C01778=1030.440,193.535,-110.316,169.514,44.801,158.470
C01779=1030.433,193.286,-110.292,169.510,44.803,158.470
C01780=1030.427,193.037,-110.268,169.506,44.804,158.470
C01781=1030.422,192.789,-110.244,169.503,44.807,158.470
C01782=1030.415,192.540,-110.220,169.500,44.809,158.470
C01783=1030.410,192.291,-110.196,169.497,44.811,158.470
C01784=1030.403,192.042,-110.171,169.493,44.812,158.470
C01785=1030.398,191.794,-110.147,169.489,44.814,158.471
C01786=1030.391,191.545,-110.123,169.486,44.817,158.471
C01787=1030.386,191.296,-110.099,169.483,44.818,158.471
C01788=1030.380,191.048,-110.075,169.479,44.820,158.471
C01789=1030.374,190.799,-110.051,169.476,44.822,158.471
C01790=1030.368,190.550,-110.027,169.472,44.824,158.471
C01791=1030.361,190.301,-110.003,169.469,44.826,158.471
C01792=1030.356,190.053,-109.979,169.466,44.828,158.471
C01793=1030.349,189.804,-109.955,169.462,44.830,158.471
C01794=1030.344,189.555,-109.930,169.459,44.831,158.471
C01795=1030.338,189.306,-109.907,169.455,44.834,158.471
C01796=1030.332,189.057,-109.883,169.451,44.836,158.471
C01797=1030.325,188.774,-109.856,169.448,44.838,158.471
C01798=1030.319,188.491,-109.828,169.444,44.840,158.471
C01799=1030.312,188.207,-109.801,169.441,44.842,158.471
C01800=1030.305,187.923,-109.774,169.436,44.845,158.471
C01801=1030.299,187.675,-109.750,169.433,44.847,158.472
C01802=1030.293,187.426,-109.725,169.430,44.848,158.472
C01803=1030.288,187.177,-109.702,169.426,44.850,158.472
C01804=1030.282,186.929,-109.679,169.423,44.852,158.472
C01805=1030.276,186.679,-109.654,169.420,44.854,158.472
C01806=1030.270,186.431,-109.631,169.416,44.856,158.472
C01807=1030.264,186.182,-109.606,169.413,44.858,158.472
C01808=1030.258,185.933,-109.583,169.409,44.860,158.472
C01809=1030.252,185.685,-109.559,169.407,44.862,158.472
C01810=1030.247,185.436,-109.535,169.403,44.864,158.472
C01811=1030.240,185.186,-109.512,169.399,44.866,158.472
C01812=1030.235,184.938,-109.487,169.396,44.868,158.472
C01813=1030.229,184.689,-109.464,169.393,44.870,158.472
C01814=1030.223,184.440,-109.439,169.390,44.872,158.472
C01815=1030.217,184.191,-109.416,169.386,44.874,158.472
C01816=1030.211,183.943,-109.393,169.383,44.875,158.473
C01817=1030.206,183.694,-109.369,169.380,44.878,158.473
C01818=1030.200,183.445,-109.345,169.376,44.880,158.473
C01819=1030.194,183.196,-109.321,169.373,44.881,158.473
C01820=1030.189,182.947,-109.298,169.370,44.883,158.473
C01821=1030.183,182.699,-109.274,169.366,44.885,158.473
C01822=1030.176,182.449,-109.251,169.363,44.888,158.473
C01823=1030.170,182.201,-109.227,169.360,44.890,158.473
C01824=1030.164,181.953,-109.205,169.357,44.892,158.473
C01825=1030.158,181.703,-109.182,169.353,44.895,158.473
C01826=1030.152,181.455,-109.158,169.350,44.897,158.474
C01827=1030.146,181.206,-109.135,169.347,44.899,158.474
C01828=1030.139,180.956,-109.112,169.344,44.901,158.474
C01829=1030.133,180.708,-109.088,169.340,44.903,158.474
C01830=1030.127,180.459,-109.066,169.336,44.905,158.474
C01831=1030.121,180.210,-109.042,169.333,44.907,158.474
C01832=1030.115,179.962,-109.019,169.330,44.909,158.474
C01833=1030.109,179.713,-108.996,169.327,44.912,158.474
C01834=1030.103,179.464,-108.973,169.323,44.914,158.475
C01835=1030.096,179.215,-108.949,169.320,44.916,158.475
C01836=1030.090,178.966,-108.926,169.317,44.918,158.475
C01837=1030.084,178.717,-108.903,169.314,44.921,158.475
C01838=1030.079,178.468,-108.880,169.310,44.923,158.475
C01839=1030.072,178.219,-108.856,169.308,44.925,158.475
C01840=1030.065,177.971,-108.834,169.304,44.927,158.475
C01841=1030.060,177.722,-108.811,169.301,44.930,158.475
C01842=1030.054,177.473,-108.788,169.297,44.932,158.476
C01843=1030.048,177.223,-108.765,169.295,44.934,158.476
C01844=1030.042,176.975,-108.741,169.291,44.936,158.476
C01845=1030.035,176.727,-108.719,169.288,44.938,158.476
C01846=1030.029,176.478,-108.696,169.285,44.940,158.476
C01847=1030.024,176.229,-108.673,169.281,44.942,158.476
C01848=1030.017,175.979,-108.650,169.278,44.945,158.476
C01849=1030.012,175.730,-108.627,169.276,44.947,158.476
C01850=1030.005,175.482,-108.604,169.272,44.949,158.477
C01851=1029.999,175.233,-108.581,169.268,44.951,158.477
C01852=1029.993,174.984,-108.558,169.265,44.954,158.477
C01853=1029.988,174.736,-108.535,169.262,44.956,158.477
C01854=1029.981,174.486,-108.512,169.259,44.958,158.477
C01855=1029.975,174.237,-108.489,169.255,44.961,158.477
C01856=1029.969,173.989,-108.466,169.253,44.963,158.477
C01857=1029.963,173.740,-108.443,169.249,44.965,158.477
C01858=1029.958,173.491,-108.420,169.247,44.967,158.478
C01859=1029.951,173.242,-108.398,169.243,44.969,158.478
C01860=1029.945,172.993,-108.375,169.240,44.971,158.478
C01861=1029.938,172.709,-108.349,169.236,44.974,158.478
C01862=1029.931,172.426,-108.322,169.233,44.976,158.478
C01863=1029.926,172.142,-108.296,169.229,44.979,158.478
C01864=1029.918,171.858,-108.270,169.226,44.981,158.478
C01865=1029.912,171.609,-108.248,169.222,44.983,158.478
C01866=1029.906,171.360,-108.225,169.219,44.986,158.479
C01867=1029.900,171.111,-108.202,169.216,44.988,158.479
C01868=1029.895,170.862,-108.179,169.213,44.990,158.479
C01869=1029.888,170.614,-108.156,169.210,44.992,158.479
C01870=1029.882,170.365,-108.133,169.207,44.994,158.479
C01871=1029.877,170.116,-108.110,169.203,44.996,158.479
C01872=1029.870,169.866,-108.087,169.201,44.999,158.480
C01873=1029.864,169.618,-108.065,169.197,45.001,158.480
C01874=1029.859,169.368,-108.043,169.195,45.003,158.480
C01875=1029.853,169.119,-108.020,169.191,45.005,158.480
C01876=1029.847,168.871,-107.997,169.188,45.008,158.480
C01877=1029.841,168.622,-107.974,169.185,45.010,158.480
C01878=1029.835,168.373,-107.951,169.182,45.012,158.480
C01879=1029.829,168.124,-107.928,169.179,45.014,158.480
C01880=1029.823,167.875,-107.906,169.176,45.017,158.480
C01881=1029.818,167.626,-107.883,169.173,45.019,158.481
C01882=1029.812,167.377,-107.861,169.170,45.021,158.481
C01883=1029.806,167.128,-107.838,169.166,45.023,158.481
C01884=1029.801,166.880,-107.815,169.164,45.025,158.481
C01885=1029.794,166.632,-107.793,169.160,45.028,158.481
C01886=1029.788,166.383,-107.770,169.158,45.030,158.481
C01887=1029.783,166.134,-107.747,169.154,45.032,158.481
C01888=1029.777,165.884,-107.725,169.152,45.034,158.482
C01889=1029.771,165.636,-107.703,169.148,45.037,158.482
C01890=1029.765,165.387,-107.680,169.146,45.039,158.482
C01891=1029.759,165.138,-107.657,169.142,45.041,158.482
C01892=1029.754,164.888,-107.634,169.140,45.043,158.482
C01893=1029.747,164.640,-107.612,169.136,45.045,158.482
C01894=1029.742,164.391,-107.589,169.133,45.047,158.482
C01895=1029.736,164.142,-107.566,169.130,45.050,158.483
C01896=1029.731,163.892,-107.544,169.128,45.052,158.483
C01897=1029.725,163.645,-107.522,169.124,45.054,158.483
C01898=1029.719,163.396,-107.499,169.121,45.056,158.483
C01899=1029.714,163.146,-107.477,169.118,45.058,158.483
C01900=1029.707,162.898,-107.454,169.116,45.061,158.483
C01901=1029.701,162.649,-107.432,169.112,45.063,158.483
C01902=1029.696,162.399,-107.409,169.110,45.065,158.484
C01903=1029.690,162.150,-107.386,169.106,45.067,158.484
C01904=1029.684,161.902,-107.364,169.103,45.069,158.484
C01905=1029.679,161.653,-107.342,169.100,45.071,158.484
C01906=1029.673,161.404,-107.319,169.098,45.074,158.484
C01907=1029.667,161.155,-107.296,169.094,45.076,158.484
C01908=1029.661,160.906,-107.275,169.092,45.078,158.484
C01909=1029.656,160.657,-107.252,169.088,45.080,158.484
C01910=1029.650,160.407,-107.229,169.085,45.082,158.485
C01911=1029.644,160.160,-107.207,169.082,45.085,158.485
C01912=1029.639,159.911,-107.185,169.080,45.087,158.485
C01913=1029.633,159.661,-107.162,169.076,45.089,158.485
C01914=1029.627,159.413,-107.140,169.073,45.091,158.485
C01915=1029.621,159.163,-107.118,169.070,45.094,158.485
C01916=1029.615,158.914,-107.096,169.068,45.096,158.486
C01917=1029.609,158.666,-107.074,169.064,45.099,158.486
C01918=1029.603,158.417,-107.052,169.062,45.101,158.486
C01919=1029.597,158.168,-107.029,169.058,45.103,158.486
C01920=1029.591,157.919,-107.008,169.056,45.106,158.486
C01921=1029.585,157.669,-106.986,169.052,45.108,158.486
C01922=1029.579,157.420,-106.963,169.050,45.110,158.487
C01923=1029.573,157.171,-106.942,169.046,45.113,158.487
C01924=1029.568,156.923,-106.920,169.044,45.115,158.487
C01925=1029.558,156.533,-106.886,169.039,45.118,158.487
C01926=1029.548,156.143,-106.851,169.035,45.122,158.487
C01927=1029.539,155.754,-106.817,169.030,45.126,158.488
C01928=1029.530,155.363,-106.782,169.026,45.130,158.488
C01929=1029.525,155.115,-106.761,169.022,45.132,158.488
C01930=1029.518,154.866,-106.739,169.020,45.134,158.488
C01931=1029.513,154.617,-106.716,169.016,45.137,158.489
C01932=1029.506,154.368,-106.695,169.014,45.139,158.489
C01933=1029.500,154.118,-106.673,169.010,45.142,158.489
C01934=1029.495,153.870,-106.652,169.008,45.144,158.489
C01935=1029.489,153.620,-106.629,169.004,45.147,158.489
C01936=1029.483,153.372,-106.607,169.002,45.149,158.489
C01937=1029.477,153.123,-106.585,168.999,45.151,158.490
C01938=1029.471,152.874,-106.564,168.996,45.153,158.490
C01939=1029.465,152.625,-106.543,168.994,45.155,158.490
C01940=1029.459,152.376,-106.521,168.990,45.158,158.490
C01941=1029.450,151.983,-106.487,168.986,45.162,158.490
C01942=1029.440,151.591,-106.452,168.981,45.166,158.491
C01943=1029.431,151.198,-106.419,168.977,45.170,158.491
C01944=1029.422,150.805,-106.384,168.972,45.174,158.491
C01945=1029.416,150.556,-106.362,168.969,45.176,158.491
C01946=1029.410,150.308,-106.340,168.966,45.178,158.492
C01947=1029.404,150.059,-106.319,168.964,45.180,158.492
C01948=1029.398,149.810,-106.297,168.960,45.183,158.492
C01949=1029.392,149.561,-106.276,168.958,45.185,158.492
C01950=1029.386,149.312,-106.254,168.955,45.188,158.492
C01951=1029.380,149.063,-106.232,168.952,45.190,158.493
C01952=1029.374,148.814,-106.211,168.950,45.193,158.493
C01953=1029.368,148.565,-106.190,168.946,45.195,158.493
C01954=1029.362,148.316,-106.168,168.944,45.198,158.493
C01955=1029.356,148.068,-106.147,168.940,45.200,158.493
C01956=1029.351,147.818,-106.124,168.938,45.202,158.494
C01957=1029.345,147.569,-106.103,168.935,45.204,158.494
C01958=1029.339,147.320,-106.082,168.932,45.207,158.494
C01959=1029.333,147.071,-106.061,168.929,45.209,158.494
C01960=1029.327,146.821,-106.039,168.926,45.212,158.494
C01961=1029.321,146.573,-106.018,168.924,45.214,158.494
C01962=1029.315,146.324,-105.996,168.920,45.217,158.495
C01963=1029.308,146.075,-105.975,168.918,45.219,158.495
C01964=1029.303,145.826,-105.954,168.916,45.222,158.495
C01965=1029.297,145.577,-105.932,168.912,45.224,158.495
C01966=1029.291,145.328,-105.911,168.910,45.226,158.495
C01967=1029.285,145.079,-105.890,168.906,45.229,158.496
C01968=1029.279,144.829,-105.868,168.904,45.231,158.496
C01969=1029.273,144.580,-105.847,168.901,45.234,158.496
C01970=1029.267,144.332,-105.826,168.898,45.237,158.496
C01971=1029.260,144.083,-105.804,168.896,45.239,158.496
C01972=1029.255,143.834,-105.784,168.892,45.242,158.497
C01973=1029.249,143.585,-105.762,168.890,45.244,158.497
C01974=1029.243,143.335,-105.741,168.887,45.247,158.497
C01975=1029.237,143.087,-105.719,168.884,45.249,158.497
C01976=1029.231,142.837,-105.699,168.881,45.251,158.497
C01977=1029.225,142.589,-105.678,168.878,45.254,158.498
C01978=1029.219,142.340,-105.656,168.876,45.256,158.498
C01979=1029.213,142.090,-105.634,168.873,45.259,158.498
C01980=1029.208,141.841,-105.614,168.870,45.262,158.498
C01981=1029.201,141.592,-105.592,168.867,45.264,158.498
C01982=1029.195,141.344,-105.572,168.864,45.266,158.499
C01983=1029.189,141.094,-105.551,168.862,45.268,158.499
C01984=1029.184,140.846,-105.529,168.859,45.271,158.499
C01985=1029.176,140.561,-105.505,168.855,45.274,158.499
C01986=1029.170,140.276,-105.480,168.853,45.277,158.500
C01987=1029.163,139.991,-105.457,168.850,45.280,158.500
C01988=1029.157,139.707,-105.433,168.846,45.283,158.500
C01989=1029.151,139.458,-105.411,168.844,45.285,158.500
C01990=1029.145,139.209,-105.391,168.841,45.287,158.500
C01991=1029.139,138.959,-105.369,168.838,45.289,158.501
C01992=1029.133,138.711,-105.349,168.835,45.292,158.501
C01993=1029.127,138.461,-105.327,168.832,45.295,158.501
C01994=1029.121,138.213,-105.306,168.830,45.297,158.501
C01995=1029.115,137.963,-105.286,168.827,45.300,158.501
C01996=1029.109,137.715,-105.264,168.824,45.302,158.502
C01997=1029.103,137.465,-105.244,168.822,45.304,158.502
C01998=1029.097,137.217,-105.223,168.818,45.307,158.502
C01999=1029.091,136.967,-105.202,168.816,45.310,158.502
C02000=1029.086,136.719,-105.181,168.813,45.312,158.502
C02001=1029.079,136.469,-105.160,168.810,45.315,158.503
C02002=1029.074,136.221,-105.139,168.808,45.318,158.503
C02003=1029.067,135.971,-105.119,168.805,45.320,158.503
C02004=1029.061,135.722,-105.097,168.802,45.322,158.503
C02005=1029.056,135.473,-105.077,168.800,45.325,158.504
C02006=1029.050,135.224,-105.057,168.797,45.328,158.504
C02007=1029.043,134.975,-105.035,168.794,45.330,158.504
C02008=1029.037,134.726,-105.015,168.791,45.333,158.504
C02009=1029.031,134.477,-104.993,168.789,45.335,158.504
C02010=1029.026,134.228,-104.973,168.786,45.337,158.505
C02011=1029.019,133.978,-104.952,168.783,45.340,158.505
C02012=1029.014,133.729,-104.931,168.780,45.343,158.505
C02013=1029.007,133.480,-104.911,168.778,45.345,158.505
C02014=1029.002,133.231,-104.890,168.775,45.348,158.505
C02015=1028.996,132.983,-104.870,168.772,45.351,158.506
C02016=1028.990,132.733,-104.849,168.770,45.353,158.506
C02017=1028.983,132.485,-104.828,168.766,45.355,158.506
C02018=1028.978,132.235,-104.807,168.764,45.358,158.506
C02019=1028.972,131.986,-104.787,168.762,45.360,158.506
C02020=1028.965,131.737,-104.766,168.758,45.363,158.507
C02021=1028.960,131.488,-104.745,168.756,45.366,158.507
C02022=1028.954,131.239,-104.725,168.754,45.368,158.507
C02023=1028.948,130.990,-104.703,168.750,45.370,158.507
C02024=1028.942,130.741,-104.683,168.748,45.373,158.508
C02025=1028.936,130.491,-104.663,168.745,45.375,158.508
C02026=1028.930,130.242,-104.643,168.742,45.378,158.508
C02027=1028.924,129.993,-104.623,168.740,45.381,158.508
C02028=1028.918,129.744,-104.601,168.738,45.383,158.509
C02029=1028.912,129.495,-104.581,168.734,45.386,158.509
C02030=1028.905,129.246,-104.561,168.732,45.389,158.509
C02031=1028.899,128.997,-104.541,168.729,45.392,158.509
C02032=1028.894,128.747,-104.520,168.726,45.394,158.509
C02033=1028.888,128.498,-104.500,168.724,45.396,158.510
C02034=1028.882,128.250,-104.480,168.721,45.399,158.510
C02035=1028.875,128.000,-104.460,168.718,45.402,158.510
C02036=1028.869,127.752,-104.438,168.716,45.405,158.510
C02037=1028.863,127.503,-104.418,168.713,45.408,158.511
C02038=1028.857,127.253,-104.398,168.710,45.410,158.511
C02039=1028.851,127.004,-104.378,168.708,45.412,158.511
C02040=1028.844,126.755,-104.358,168.705,45.415,158.511
C02041=1028.839,126.506,-104.337,168.702,45.418,158.512
C02042=1028.833,126.257,-104.317,168.700,45.420,158.512
C02043=1028.826,126.007,-104.297,168.696,45.423,158.512
C02044=1028.820,125.759,-104.277,168.694,45.425,158.512
C02045=1028.815,125.510,-104.256,168.691,45.428,158.512
C02046=1028.809,125.260,-104.236,168.689,45.431,158.513
C02047=1028.803,125.011,-104.216,168.686,45.434,158.513
C02048=1028.797,124.762,-104.196,168.684,45.436,158.513
C02049=1028.790,124.477,-104.172,168.681,45.439,158.514
C02050=1028.782,124.193,-104.150,168.677,45.442,158.514
C02051=1028.776,123.908,-104.127,168.674,45.445,158.514
C02052=1028.769,123.624,-104.104,168.671,45.448,158.514
C02053=1028.763,123.374,-104.083,168.669,45.451,158.515
C02054=1028.757,123.125,-104.063,168.666,45.453,158.515
C02055=1028.751,122.876,-104.043,168.663,45.456,158.515
C02056=1028.744,122.627,-104.023,168.661,45.459,158.515
C02057=1028.738,122.378,-104.003,168.658,45.461,158.515
C02058=1028.733,122.129,-103.982,168.655,45.464,158.516
C02059=1028.727,121.880,-103.962,168.653,45.466,158.516
C02060=1028.721,121.630,-103.943,168.650,45.469,158.516
C02061=1028.715,121.381,-103.923,168.648,45.471,158.516
C02062=1028.710,121.132,-103.902,168.645,45.474,158.517
C02063=1028.703,120.882,-103.882,168.642,45.477,158.517
C02064=1028.697,120.633,-103.862,168.640,45.479,158.517
C02065=1028.691,120.385,-103.842,168.637,45.482,158.517
C02066=1028.685,120.136,-103.822,168.634,45.484,158.517
C02067=1028.680,119.887,-103.801,168.632,45.487,158.518
C02068=1028.674,119.637,-103.782,168.630,45.489,158.518
C02069=1028.668,119.388,-103.762,168.626,45.492,158.518
C02070=1028.662,119.139,-103.742,168.624,45.494,158.518
C02071=1028.656,118.890,-103.722,168.621,45.497,158.519
C02072=1028.649,118.641,-103.701,168.619,45.500,158.519
C02073=1028.644,118.392,-103.681,168.616,45.503,158.519
C02074=1028.638,118.143,-103.661,168.613,45.505,158.519
C02075=1028.632,117.893,-103.642,168.611,45.507,158.520
C02076=1028.626,117.644,-103.622,168.609,45.510,158.520
C02077=1028.619,117.395,-103.601,168.606,45.513,158.520
C02078=1028.614,117.146,-103.581,168.603,45.515,158.520
C02079=1028.609,116.896,-103.562,168.601,45.518,158.520
C02080=1028.603,116.648,-103.542,168.598,45.520,158.521
C02081=1028.597,116.399,-103.522,168.595,45.523,158.521
C02082=1028.591,116.150,-103.502,168.593,45.525,158.521
C02083=1028.584,115.900,-103.481,168.590,45.528,158.521
C02084=1028.579,115.651,-103.462,168.588,45.531,158.522
C02085=1028.573,115.402,-103.442,168.585,45.533,158.522
C02086=1028.567,115.153,-103.422,168.582,45.535,158.522
C02087=1028.561,114.904,-103.402,168.580,45.538,158.522
C02088=1028.555,114.655,-103.382,168.578,45.541,158.523
C02089=1028.550,114.406,-103.362,168.574,45.544,158.523
C02090=1028.543,114.156,-103.342,168.572,45.546,158.523
C02091=1028.538,113.907,-103.322,168.570,45.548,158.523
C02092=1028.532,113.658,-103.302,168.567,45.551,158.523
C02093=1028.526,113.409,-103.282,168.565,45.553,158.524
C02094=1028.520,113.160,-103.263,168.562,45.556,158.524
C02095=1028.515,112.911,-103.243,168.559,45.559,158.524
C02096=1028.509,112.661,-103.223,168.557,45.561,158.524
C02097=1028.502,112.412,-103.204,168.555,45.564,158.525
C02098=1028.496,112.163,-103.184,168.551,45.566,158.525
C02099=1028.490,111.914,-103.164,168.549,45.569,158.525
C02100=1028.484,111.665,-103.145,168.547,45.572,158.525
C02101=1028.478,111.415,-103.125,168.544,45.574,158.526
C02102=1028.472,111.167,-103.105,168.541,45.577,158.526
C02103=1028.467,110.917,-103.086,168.539,45.580,158.526
C02104=1028.461,110.668,-103.066,168.536,45.582,158.526
C02105=1028.455,110.419,-103.047,168.534,45.585,158.526
C02106=1028.449,110.169,-103.027,168.531,45.588,158.527
C02107=1028.442,109.920,-103.008,168.528,45.590,158.527
C02108=1028.436,109.671,-102.988,168.526,45.593,158.527
C02109=1028.430,109.422,-102.969,168.524,45.596,158.527
C02110=1028.425,109.173,-102.949,168.521,45.599,158.528
C02111=1028.418,108.924,-102.930,168.518,45.601,158.528
C02112=1028.412,108.675,-102.911,168.516,45.604,158.528
C02113=1028.405,108.390,-102.889,168.513,45.607,158.528
C02114=1028.398,108.105,-102.866,168.509,45.610,158.529
C02115=1028.391,107.820,-102.844,168.507,45.613,158.529
C02116=1028.385,107.535,-102.822,168.504,45.616,158.529
C02117=1028.378,107.285,-102.803,168.502,45.619,158.530
C02118=1028.372,107.037,-102.783,168.499,45.622,158.530
C02119=1028.366,106.787,-102.764,168.496,45.624,158.530
C02120=1028.360,106.538,-102.745,168.494,45.627,158.530
C02121=1028.354,106.289,-102.725,168.492,45.630,158.531
C02122=1028.348,106.040,-102.706,168.488,45.632,158.531
C02123=1028.342,105.790,-102.687,168.486,45.635,158.531
C02124=1028.336,105.542,-102.667,168.484,45.637,158.531
C02125=1028.330,105.293,-102.648,168.481,45.640,158.532
C02126=1028.324,105.043,-102.629,168.478,45.643,158.532
C02127=1028.318,104.794,-102.609,168.476,45.646,158.532
C02128=1028.312,104.545,-102.590,168.474,45.648,158.532
C02129=1028.306,104.296,-102.571,168.471,45.651,158.533
C02130=1028.300,104.047,-102.551,168.468,45.654,158.533
C02131=1028.294,103.797,-102.532,168.466,45.656,158.533
C02132=1028.288,103.548,-102.513,168.463,45.659,158.533
C02133=1028.282,103.299,-102.494,168.461,45.661,158.533
C02134=1028.276,103.050,-102.474,168.459,45.664,158.534
C02135=1028.270,102.801,-102.456,168.455,45.667,158.534
C02136=1028.264,102.552,-102.436,168.453,45.670,158.534
C02137=1028.258,102.302,-102.417,168.451,45.672,158.534
C02138=1028.253,102.053,-102.398,168.448,45.674,158.535
C02139=1028.246,101.804,-102.378,168.445,45.677,158.535
C02140=1028.240,101.555,-102.359,168.443,45.680,158.535
C02141=1028.235,101.305,-102.340,168.441,45.683,158.535
C02142=1028.228,101.056,-102.321,168.438,45.685,158.536
C02143=1028.222,100.807,-102.302,168.436,45.688,158.536
C02144=1028.216,100.558,-102.282,168.432,45.690,158.536
C02145=1028.210,100.309,-102.263,168.430,45.693,158.536
C02146=1028.204,100.059,-102.244,168.428,45.696,158.537
C02147=1028.199,99.810,-102.225,168.426,45.698,158.537
C02148=1028.192,99.561,-102.206,168.423,45.701,158.537
C02149=1028.186,99.311,-102.187,168.420,45.704,158.537
C02150=1028.180,99.062,-102.168,168.418,45.707,158.538
C02151=1028.174,98.813,-102.149,168.416,45.709,158.538
C02152=1028.168,98.564,-102.131,168.413,45.712,158.538
C02153=1028.162,98.315,-102.112,168.410,45.715,158.538
C02154=1028.156,98.065,-102.093,168.408,45.718,158.539
C02155=1028.150,97.817,-102.074,168.406,45.720,158.539
C02156=1028.144,97.567,-102.055,168.403,45.723,158.539
C02157=1028.138,97.318,-102.036,168.400,45.726,158.539
C02158=1028.131,97.069,-102.018,168.398,45.729,158.540
C02159=1028.126,96.820,-101.999,168.395,45.731,158.540
C02160=1028.119,96.571,-101.980,168.393,45.734,158.540
C02161=1028.114,96.321,-101.961,168.391,45.736,158.540
C02162=1028.107,96.072,-101.942,168.387,45.739,158.541
C02163=1028.102,95.823,-101.923,168.385,45.742,158.541
C02164=1028.095,95.573,-101.904,168.383,45.745,158.541
C02165=1028.089,95.324,-101.885,168.381,45.747,158.541
C02166=1028.083,95.075,-101.866,168.377,45.750,158.542
C02167=1028.077,94.826,-101.848,168.375,45.753,158.542
C02168=1028.072,94.577,-101.829,168.373,45.756,158.542
C02169=1028.065,94.328,-101.810,168.370,45.758,158.542
C02170=1028.059,94.078,-101.792,168.368,45.761,158.543
C02171=1028.053,93.829,-101.773,168.365,45.764,158.543
C02172=1028.047,93.580,-101.754,168.363,45.767,158.543
C02173=1028.041,93.330,-101.735,168.360,45.769,158.543
C02174=1028.035,93.081,-101.716,168.358,45.771,158.544
C02175=1028.029,92.833,-101.698,168.356,45.774,158.544
C02176=1028.023,92.583,-101.679,168.352,45.777,158.544
C02177=1028.016,92.298,-101.658,168.350,45.780,158.544
C02178=1028.009,92.013,-101.636,168.347,45.783,158.545
C02179=1028.003,91.729,-101.615,168.344,45.786,158.545
C02180=1027.996,91.443,-101.594,168.342,45.790,158.545
C02181=1027.990,91.194,-101.575,168.339,45.792,158.545
C02182=1027.983,90.945,-101.556,168.336,45.795,158.546
C02183=1027.977,90.696,-101.537,168.334,45.797,158.546
C02184=1027.972,90.447,-101.518,168.331,45.800,158.546
C02185=1027.966,90.197,-101.501,168.329,45.803,158.546
C02186=1027.960,89.948,-101.481,168.327,45.805,158.547
C02187=1027.954,89.699,-101.463,168.324,45.808,158.547
C02188=1027.947,89.450,-101.444,168.321,45.811,158.547
C02189=1027.941,89.200,-101.426,168.319,45.814,158.547
C02190=1027.935,88.951,-101.408,168.317,45.817,158.548
C02191=1027.930,88.702,-101.389,168.315,45.819,158.548
C02192=1027.924,88.452,-101.371,168.311,45.822,158.548
C02193=1027.917,88.203,-101.352,168.309,45.825,158.548
C02194=1027.911,87.954,-101.333,168.307,45.828,158.549
C02195=1027.905,87.704,-101.315,168.305,45.830,158.549
C02196=1027.899,87.456,-101.297,168.301,45.833,158.549
C02197=1027.893,87.206,-101.279,168.299,45.836,158.550
C02198=1027.886,86.957,-101.261,168.297,45.839,158.550
C02199=1027.880,86.708,-101.242,168.294,45.841,158.550
C02200=1027.874,86.458,-101.224,168.291,45.844,158.550
C02201=1027.868,86.210,-101.206,168.289,45.847,158.551
C02202=1027.862,85.960,-101.187,168.287,45.850,158.551
C02203=1027.856,85.710,-101.168,168.284,45.852,158.551
C02204=1027.850,85.461,-101.150,168.282,45.855,158.551
C02205=1027.844,85.212,-101.132,168.279,45.858,158.552
C02206=1027.838,84.963,-101.114,168.277,45.861,158.552
C02207=1027.832,84.713,-101.096,168.274,45.864,158.552
C02208=1027.825,84.464,-101.077,168.272,45.866,158.552
C02209=1027.820,84.215,-101.059,168.269,45.869,158.553
C02210=1027.813,83.966,-101.041,168.267,45.872,158.553
C02211=1027.807,83.716,-101.023,168.264,45.875,158.553
C02212=1027.801,83.467,-101.004,168.262,45.877,158.553
C02213=1027.795,83.219,-100.986,168.260,45.880,158.554
C02214=1027.789,82.969,-100.967,168.256,45.882,158.554
C02215=1027.783,82.720,-100.949,168.254,45.885,158.554
C02216=1027.777,82.470,-100.931,168.252,45.888,158.554
C02217=1027.771,82.222,-100.913,168.249,45.890,158.555
C02218=1027.765,81.972,-100.895,168.247,45.893,158.555
C02219=1027.759,81.722,-100.877,168.245,45.896,158.555
C02220=1027.753,81.474,-100.858,168.242,45.899,158.555
C02221=1027.747,81.224,-100.840,168.239,45.902,158.556
C02222=1027.740,80.975,-100.822,168.237,45.904,158.556
C02223=1027.734,80.725,-100.804,168.235,45.907,158.556
C02224=1027.728,80.477,-100.786,168.233,45.910,158.556
C02225=1027.722,80.227,-100.768,168.229,45.913,158.557
C02226=1027.716,79.978,-100.749,168.227,45.915,158.557
C02227=1027.710,79.729,-100.731,168.225,45.918,158.557
C02228=1027.705,79.479,-100.713,168.222,45.920,158.557
C02229=1027.699,79.230,-100.694,168.220,45.923,158.557
C02230=1027.693,78.980,-100.677,168.218,45.926,158.558
C02231=1027.687,78.731,-100.658,168.215,45.929,158.558
C02232=1027.681,78.482,-100.641,168.212,45.931,158.558
C02233=1027.675,78.233,-100.623,168.210,45.934,158.558
C02234=1027.669,77.983,-100.604,168.208,45.937,158.559
C02235=1027.663,77.734,-100.586,168.206,45.939,158.559
C02236=1027.657,77.485,-100.568,168.202,45.942,158.559
C02237=1027.651,77.236,-100.550,168.200,45.945,158.559
C02238=1027.645,76.987,-100.532,168.198,45.948,158.560
C02239=1027.639,76.737,-100.514,168.196,45.951,158.560
C02240=1027.632,76.488,-100.496,168.193,45.953,158.560
C02241=1027.625,76.203,-100.476,168.190,45.956,158.560
C02242=1027.618,75.917,-100.456,168.187,45.959,158.561
C02243=1027.611,75.633,-100.436,168.185,45.963,158.561
C02244=1027.604,75.348,-100.415,168.181,45.966,158.561
C02245=1027.599,75.098,-100.397,168.179,45.968,158.562
C02246=1027.592,74.849,-100.379,168.177,45.971,158.562
C02247=1027.586,74.600,-100.361,168.174,45.974,158.562
C02248=1027.580,74.351,-100.344,168.171,45.977,158.562
C02249=1027.574,74.101,-100.326,168.169,45.979,158.563
C02250=1027.568,73.852,-100.308,168.167,45.982,158.563
C02251=1027.562,73.603,-100.290,168.165,45.985,158.563
C02252=1027.556,73.353,-100.272,168.161,45.988,158.563
C02253=1027.549,73.105,-100.255,168.159,45.991,158.564
C02254=1027.543,72.855,-100.237,168.157,45.993,158.564
C02255=1027.538,72.606,-100.219,168.155,45.996,158.564
C02256=1027.532,72.356,-100.201,168.152,45.999,158.564
C02257=1027.525,72.107,-100.184,168.149,46.002,158.565
C02258=1027.519,71.858,-100.166,168.147,46.004,158.565
C02259=1027.513,71.608,-100.148,168.145,46.007,158.565
C02260=1027.507,71.359,-100.130,168.142,46.010,158.565
C02261=1027.500,71.110,-100.113,168.140,46.013,158.566
C02262=1027.495,70.861,-100.095,168.137,46.016,158.566
C02263=1027.489,70.611,-100.077,168.135,46.018,158.566
C02264=1027.483,70.361,-100.060,168.132,46.021,158.566
C02265=1027.476,70.113,-100.043,168.130,46.024,158.567
C02266=1027.470,69.863,-100.025,168.128,46.026,158.567
C02267=1027.465,69.614,-100.007,168.125,46.029,158.567
C02268=1027.459,69.364,-99.989,168.122,46.032,158.567
C02269=1027.452,69.115,-99.972,168.120,46.035,158.568
C02270=1027.446,68.866,-99.954,168.118,46.038,158.568
C02271=1027.441,68.617,-99.937,168.116,46.040,158.568
C02272=1027.434,68.367,-99.919,168.112,46.043,158.568
C02273=1027.428,68.118,-99.902,168.110,46.046,158.569
C02274=1027.422,67.868,-99.884,168.108,46.049,158.569
C02275=1027.416,67.620,-99.867,168.106,46.052,158.569
C02276=1027.410,67.370,-99.849,168.103,46.054,158.569
C02277=1027.404,67.121,-99.832,168.100,46.057,158.570
C02278=1027.398,66.872,-99.814,168.098,46.060,158.570
C02279=1027.392,66.622,-99.796,168.095,46.063,158.570
C02280=1027.385,66.373,-99.779,168.093,46.065,158.570
C02281=1027.380,66.124,-99.762,168.091,46.068,158.571
C02282=1027.373,65.875,-99.744,168.088,46.071,158.571
C02283=1027.367,65.626,-99.727,168.085,46.074,158.571
C02284=1027.361,65.375,-99.710,168.083,46.077,158.571
C02285=1027.355,65.126,-99.692,168.081,46.079,158.572
C02286=1027.348,64.877,-99.675,168.078,46.082,158.572
C02287=1027.343,64.628,-99.658,168.075,46.085,158.572
C02288=1027.337,64.378,-99.640,168.073,46.088,158.572
C02289=1027.330,64.130,-99.623,168.071,46.091,158.573
C02290=1027.324,63.880,-99.605,168.069,46.093,158.573
C02291=1027.318,63.630,-99.588,168.065,46.096,158.573
C02292=1027.312,63.381,-99.570,168.063,46.099,158.573
C02293=1027.306,63.132,-99.554,168.061,46.102,158.574
C02294=1027.299,62.883,-99.536,168.059,46.104,158.574
C02295=1027.294,62.633,-99.519,168.055,46.107,158.574
C02296=1027.287,62.383,-99.502,168.053,46.110,158.574
C02297=1027.281,62.135,-99.485,168.051,46.113,158.575
C02298=1027.274,61.885,-99.468,168.049,46.116,158.575
C02299=1027.269,61.636,-99.451,168.046,46.119,158.575
C02300=1027.262,61.386,-99.433,168.043,46.122,158.576
C02301=1027.256,61.137,-99.417,168.041,46.125,158.576
C02302=1027.250,60.888,-99.400,168.039,46.127,158.576
C02303=1027.244,60.638,-99.382,168.036,46.130,158.576
C02304=1027.238,60.389,-99.366,168.033,46.133,158.577
C02305=1027.230,60.104,-99.346,168.030,46.137,158.577
C02306=1027.222,59.819,-99.327,168.028,46.140,158.577
C02307=1027.216,59.534,-99.307,168.025,46.143,158.578
C02308=1027.208,59.248,-99.288,168.022,46.147,158.578
C02309=1027.202,59.000,-99.271,168.020,46.150,158.578
C02310=1027.196,58.749,-99.254,168.018,46.152,158.578
C02311=1027.190,58.500,-99.237,168.014,46.155,158.579
C02312=1027.184,58.252,-99.220,168.012,46.158,158.579
C02313=1027.177,58.002,-99.203,168.010,46.161,158.579
C02314=1027.172,57.753,-99.186,168.008,46.164,158.579
C02315=1027.165,57.503,-99.169,168.004,46.167,158.580
C02316=1027.159,57.254,-99.152,168.002,46.169,158.580
C02317=1027.153,57.005,-99.136,168.000,46.172,158.580
C02318=1027.146,56.755,-99.119,167.998,46.175,158.580
C02319=1027.141,56.506,-99.101,167.994,46.178,158.581
C02320=1027.135,56.257,-99.085,167.992,46.181,158.581
C02321=1027.128,56.007,-99.067,167.990,46.184,158.581
C02322=1027.122,55.758,-99.051,167.988,46.187,158.582
C02323=1027.116,55.508,-99.033,167.986,46.189,158.582
C02324=1027.110,55.259,-99.017,167.982,46.192,158.582
C02325=1027.104,55.010,-99.000,167.980,46.195,158.582
C02326=1027.097,54.760,-98.983,167.978,46.198,158.583
C02327=1027.091,54.511,-98.966,167.976,46.201,158.583
C02328=1027.086,54.262,-98.950,167.972,46.204,158.583
C02329=1027.079,54.012,-98.932,167.970,46.206,158.583
C02330=1027.073,53.763,-98.916,167.968,46.209,158.584
C02331=1027.066,53.514,-98.899,167.966,46.212,158.584
C02332=1027.061,53.264,-98.882,167.962,46.215,158.584
C02333=1027.055,53.014,-98.865,167.960,46.218,158.584
C02334=1027.048,52.766,-98.849,167.958,46.220,158.584
C02335=1027.042,52.516,-98.832,167.956,46.223,158.585
C02336=1027.036,52.267,-98.815,167.954,46.226,158.585
C02337=1027.030,52.017,-98.798,167.950,46.229,158.585
C02338=1027.024,51.769,-98.781,167.948,46.232,158.585
C02339=1027.018,51.518,-98.764,167.946,46.234,158.586
C02340=1027.012,51.269,-98.748,167.944,46.237,158.586
C02341=1027.006,51.020,-98.731,167.940,46.240,158.586
C02342=1027.000,50.770,-98.714,167.938,46.243,158.586
C02343=1026.993,50.521,-98.697,167.936,46.246,158.587
C02344=1026.987,50.272,-98.681,167.934,46.248,158.587
C02345=1026.981,50.023,-98.665,167.931,46.251,158.587
C02346=1026.975,49.773,-98.647,167.928,46.254,158.587
C02347=1026.969,49.524,-98.630,167.926,46.257,158.588
C02348=1026.963,49.274,-98.614,167.923,46.259,158.588
C02349=1026.957,49.025,-98.597,167.921,46.262,158.588
C02350=1026.951,48.775,-98.580,167.919,46.264,158.588
C02351=1026.945,48.526,-98.564,167.916,46.267,158.588
C02352=1026.939,48.277,-98.547,167.913,46.270,158.589
C02353=1026.933,48.028,-98.530,167.911,46.273,158.589
C02354=1026.927,47.778,-98.514,167.909,46.276,158.589
C02355=1026.920,47.529,-98.497,167.907,46.278,158.590
C02356=1026.915,47.279,-98.480,167.903,46.281,158.590
C02357=1026.909,47.030,-98.464,167.901,46.284,158.590
C02358=1026.903,46.781,-98.447,167.899,46.287,158.590
C02359=1026.897,46.532,-98.430,167.897,46.290,158.591
C02360=1026.890,46.282,-98.414,167.894,46.292,158.591
C02361=1026.884,46.032,-98.398,167.891,46.295,158.591
C02362=1026.879,45.783,-98.380,167.889,46.298,158.591
C02363=1026.873,45.534,-98.364,167.886,46.300,158.591
C02364=1026.867,45.285,-98.348,167.884,46.303,158.592
C02365=1026.860,45.035,-98.331,167.882,46.306,158.592
C02366=1026.854,44.786,-98.314,167.880,46.309,158.592
C02367=1026.849,44.536,-98.297,167.876,46.312,158.592
C02368=1026.843,44.287,-98.281,167.874,46.314,158.593
C02369=1026.836,44.002,-98.262,167.871,46.317,158.593
C02370=1026.829,43.716,-98.244,167.869,46.320,158.593
C02371=1026.822,43.431,-98.224,167.865,46.323,158.593
C02372=1026.815,43.145,-98.205,167.863,46.327,158.594
C02373=1026.809,42.896,-98.189,167.860,46.329,158.594
C02374=1026.803,42.647,-98.172,167.858,46.332,158.594
C02375=1026.797,42.398,-98.156,167.855,46.334,158.594
C02376=1026.791,42.148,-98.140,167.853,46.337,158.594
C02377=1026.785,41.898,-98.123,167.850,46.340,158.595
C02378=1026.779,41.649,-98.107,167.848,46.343,158.595
C02379=1026.773,41.399,-98.090,167.845,46.346,158.595
C02380=1026.767,41.150,-98.074,167.843,46.348,158.595
C02381=1026.761,40.901,-98.058,167.840,46.351,158.596
C02382=1026.755,40.651,-98.042,167.838,46.354,158.596
C02383=1026.749,40.402,-98.025,167.835,46.357,158.596
C02384=1026.742,40.153,-98.010,167.833,46.360,158.596
C02385=1026.736,39.903,-97.993,167.830,46.363,158.596
C02386=1026.730,39.654,-97.977,167.828,46.365,158.597
C02387=1026.724,39.404,-97.961,167.825,46.368,158.597
C02388=1026.718,39.155,-97.944,167.823,46.371,158.597
C02389=1026.712,38.906,-97.928,167.821,46.374,158.598
C02390=1026.706,38.656,-97.912,167.818,46.377,158.598
C02391=1026.700,38.407,-97.896,167.815,46.380,158.598
C02392=1026.694,38.158,-97.879,167.813,46.382,158.598
C02393=1026.688,37.908,-97.863,167.811,46.385,158.598
C02394=1026.681,37.659,-97.847,167.808,46.388,158.599
C02395=1026.675,37.409,-97.831,167.806,46.391,158.599
C02396=1026.669,37.160,-97.815,167.803,46.394,158.599
C02397=1026.663,36.910,-97.798,167.801,46.396,158.599
C02398=1026.657,36.660,-97.783,167.798,46.399,158.600
C02399=1026.651,36.411,-97.767,167.796,46.402,158.600
C02400=1026.645,36.162,-97.751,167.793,46.405,158.600
C02401=1026.639,35.913,-97.735,167.791,46.408,158.600
C02402=1026.632,35.664,-97.719,167.788,46.411,158.601
C02403=1026.626,35.414,-97.703,167.786,46.413,158.601
C02404=1026.621,35.164,-97.687,167.783,46.416,158.601
C02405=1026.614,34.915,-97.671,167.780,46.419,158.601
C02406=1026.608,34.666,-97.655,167.778,46.422,158.602
C02407=1026.602,34.417,-97.639,167.776,46.425,158.602
C02408=1026.596,34.167,-97.624,167.773,46.428,158.602
C02409=1026.590,33.918,-97.608,167.770,46.431,158.602
C02410=1026.583,33.668,-97.591,167.768,46.433,158.602
C02411=1026.576,33.419,-97.575,167.766,46.437,158.603
C02412=1026.571,33.169,-97.560,167.763,46.440,158.603
C02413=1026.565,32.919,-97.544,167.760,46.443,158.603
C02414=1026.558,32.670,-97.528,167.758,46.445,158.604
C02415=1026.552,32.421,-97.512,167.756,46.448,158.604
C02416=1026.546,32.171,-97.496,167.753,46.451,158.604
C02417=1026.540,31.922,-97.481,167.751,46.454,158.604
C02418=1026.534,31.672,-97.464,167.748,46.457,158.605
C02419=1026.528,31.423,-97.448,167.745,46.460,158.605
C02420=1026.522,31.173,-97.433,167.743,46.462,158.605
C02421=1026.516,30.924,-97.417,167.741,46.465,158.605
C02422=1026.509,30.675,-97.401,167.738,46.468,158.605
C02423=1026.503,30.425,-97.386,167.735,46.471,158.606
C02424=1026.497,30.176,-97.369,167.733,46.474,158.606
C02425=1026.491,29.927,-97.354,167.730,46.476,158.606
C02426=1026.486,29.677,-97.339,167.728,46.479,158.606
C02427=1026.480,29.428,-97.322,167.725,46.482,158.606
C02428=1026.473,29.179,-97.307,167.723,46.484,158.607
C02429=1026.467,28.929,-97.291,167.720,46.487,158.607
C02430=1026.461,28.680,-97.275,167.718,46.490,158.607
C02431=1026.455,28.430,-97.260,167.715,46.493,158.607
C02432=1026.449,28.181,-97.244,167.713,46.496,158.608
C02433=1026.442,27.895,-97.225,167.710,46.499,158.608
C02434=1026.435,27.610,-97.208,167.706,46.503,158.608
C02435=1026.428,27.324,-97.189,167.704,46.505,158.608
C02436=1026.421,27.039,-97.172,167.701,46.509,158.609
C02437=1026.415,26.789,-97.156,167.699,46.512,158.609
C02438=1026.408,26.540,-97.141,167.696,46.515,158.609
C02439=1026.402,26.291,-97.126,167.694,46.518,158.609
C02440=1026.396,26.041,-97.110,167.691,46.520,158.610
C02441=1026.389,25.792,-97.094,167.688,46.523,158.610
C02442=1026.384,25.542,-97.079,167.686,46.526,158.610
C02443=1026.378,25.293,-97.064,167.684,46.529,158.610
C02444=1026.372,25.043,-97.048,167.680,46.532,158.611
C02445=1026.365,24.794,-97.032,167.678,46.535,158.611
C02446=1026.359,24.545,-97.017,167.676,46.537,158.611
C02447=1026.353,24.295,-97.001,167.673,46.541,158.611
C02448=1026.346,24.046,-96.986,167.670,46.543,158.612
C02449=1026.341,23.796,-96.971,167.668,46.546,158.612
C02450=1026.334,23.547,-96.955,167.666,46.549,158.612
C02451=1026.328,23.297,-96.940,167.663,46.552,158.612
C02452=1026.322,23.048,-96.924,167.660,46.555,158.612
C02453=1026.316,22.799,-96.909,167.658,46.557,158.613
C02454=1026.310,22.549,-96.894,167.655,46.560,158.613
C02455=1026.304,22.300,-96.878,167.653,46.563,158.613
C02456=1026.297,22.050,-96.863,167.651,46.566,158.613
C02457=1026.292,21.800,-96.847,167.647,46.569,158.614
C02458=1026.285,21.551,-96.832,167.645,46.572,158.614
C02459=1026.279,21.302,-96.817,167.643,46.575,158.614
C02460=1026.274,21.052,-96.802,167.640,46.578,158.614
C02461=1026.267,20.803,-96.786,167.637,46.580,158.614
C02462=1026.261,20.553,-96.771,167.635,46.583,158.615
C02463=1026.255,20.303,-96.756,167.632,46.586,158.615
C02464=1026.248,20.054,-96.740,167.630,46.589,158.615
C02465=1026.243,19.805,-96.725,167.627,46.592,158.615
C02466=1026.237,19.555,-96.710,167.625,46.595,158.616
C02467=1026.230,19.306,-96.694,167.622,46.598,158.616
C02468=1026.224,19.056,-96.679,167.620,46.600,158.616
C02469=1026.218,18.807,-96.664,167.617,46.603,158.616
C02470=1026.212,18.558,-96.649,167.614,46.606,158.617
C02471=1026.206,18.308,-96.634,167.612,46.609,158.617
C02472=1026.200,18.059,-96.618,167.610,46.612,158.617
C02473=1026.193,17.809,-96.603,167.607,46.615,158.617
C02474=1026.187,17.560,-96.588,167.604,46.618,158.617
C02475=1026.181,17.311,-96.573,167.602,46.620,158.618
C02476=1026.176,17.061,-96.558,167.599,46.623,158.618
C02477=1026.169,16.812,-96.542,167.597,46.626,158.618
C02478=1026.163,16.562,-96.527,167.594,46.629,158.618
C02479=1026.156,16.312,-96.512,167.591,46.632,158.619
C02480=1026.150,16.063,-96.498,167.589,46.635,158.619
C02481=1026.145,15.813,-96.482,167.586,46.638,158.619
C02482=1026.138,15.564,-96.467,167.583,46.641,158.619
C02483=1026.132,15.314,-96.452,167.581,46.643,158.619
C02484=1026.126,15.066,-96.437,167.578,46.647,158.620
C02485=1026.120,14.816,-96.421,167.576,46.649,158.620
C02486=1026.114,14.566,-96.406,167.573,46.652,158.620
C02487=1026.108,14.316,-96.392,167.570,46.655,158.620
C02488=1026.102,14.067,-96.377,167.568,46.658,158.621
C02489=1026.096,13.817,-96.361,167.566,46.661,158.621
C02490=1026.090,13.568,-96.346,167.563,46.664,158.621
C02491=1026.083,13.318,-96.332,167.560,46.667,158.621
C02492=1026.078,13.069,-96.317,167.558,46.670,158.622
C02493=1026.071,12.820,-96.302,167.555,46.673,158.622
C02494=1026.065,12.570,-96.287,167.553,46.676,158.622
C02495=1026.059,12.321,-96.272,167.550,46.679,158.622
C02496=1026.052,12.072,-96.258,167.547,46.682,158.623
C02497=1026.045,11.787,-96.241,167.544,46.685,158.623
C02498=1026.038,11.504,-96.224,167.541,46.688,158.623
C02499=1026.031,11.219,-96.207,167.538,46.692,158.623
C02500=1026.024,10.936,-96.191,167.536,46.695,158.624
C02501=1026.017,10.686,-96.176,167.533,46.698,158.624
C02502=1026.011,10.436,-96.161,167.531,46.701,158.624
C02503=1026.005,10.186,-96.147,167.527,46.704,158.624
C02504=1025.999,9.937,-96.132,167.525,46.707,158.625
C02505=1025.993,9.687,-96.117,167.523,46.710,158.625
C02506=1025.986,9.438,-96.102,167.520,46.713,158.625
C02507=1025.981,9.189,-96.088,167.518,46.716,158.625
C02508=1025.974,8.939,-96.073,167.514,46.719,158.625
C02509=1025.968,8.689,-96.058,167.512,46.722,158.626
C02510=1025.962,8.440,-96.044,167.510,46.725,158.626
C02511=1025.956,8.190,-96.029,167.507,46.728,158.626
C02512=1025.949,7.941,-96.015,167.505,46.730,158.626
C02513=1025.943,7.692,-96.000,167.501,46.734,158.627
C02514=1025.937,7.442,-95.985,167.499,46.736,158.627
C02515=1025.931,7.193,-95.970,167.497,46.739,158.627
C02516=1025.925,6.943,-95.956,167.494,46.742,158.627
C02517=1025.919,6.693,-95.941,167.491,46.745,158.627
C02518=1025.913,6.444,-95.927,167.488,46.748,158.628
C02519=1025.906,6.195,-95.912,167.486,46.751,158.628
C02520=1025.900,5.945,-95.898,167.484,46.754,158.628
C02521=1025.894,5.696,-95.883,167.480,46.757,158.628
C02522=1025.888,5.446,-95.868,167.478,46.759,158.629
C02523=1025.882,5.197,-95.853,167.475,46.762,158.629
C02524=1025.876,4.947,-95.839,167.473,46.765,158.629
C02525=1025.870,4.698,-95.825,167.471,46.768,158.629
C02526=1025.863,4.448,-95.810,167.467,46.771,158.629
C02527=1025.857,4.199,-95.795,167.465,46.774,158.630
C02528=1025.851,3.949,-95.781,167.462,46.777,158.630
C02529=1025.845,3.699,-95.766,167.460,46.780,158.630
C02530=1025.839,3.451,-95.752,167.457,46.783,158.630
C02531=1025.833,3.200,-95.738,167.454,46.786,158.630
C02532=1025.827,2.951,-95.723,167.452,46.788,158.631
C02533=1025.821,2.702,-95.708,167.449,46.792,158.631
C02534=1025.815,2.452,-95.693,167.446,46.794,158.631
C02535=1025.809,2.202,-95.679,167.444,46.797,158.631
C02536=1025.803,1.953,-95.664,167.441,46.800,158.631
C02537=1025.797,1.703,-95.651,167.439,46.803,158.632
C02538=1025.790,1.454,-95.636,167.437,46.806,158.632
C02539=1025.784,1.205,-95.622,167.433,46.809,158.632
C02540=1025.778,0.955,-95.607,167.431,46.812,158.632
C02541=1025.773,0.706,-95.593,167.428,46.815,158.633
C02542=1025.766,0.456,-95.578,167.426,46.818,158.633
C02543=1025.761,0.206,-95.564,167.423,46.820,158.633
C02544=1025.754,-0.043,-95.549,167.420,46.823,158.633
C02545=1025.749,-0.293,-95.535,167.418,46.826,158.633
C02546=1025.743,-0.542,-95.520,167.414,46.829,158.633
C02547=1025.737,-0.791,-95.506,167.412,46.831,158.634
C02548=1025.731,-1.041,-95.492,167.410,46.834,158.634
C02549=1025.724,-1.290,-95.477,167.407,46.837,158.634
C02550=1025.719,-1.540,-95.464,167.405,46.840,158.634
C02551=1025.712,-1.790,-95.449,167.402,46.843,158.635
C02552=1025.707,-2.039,-95.435,167.399,46.846,158.635
C02553=1025.700,-2.289,-95.420,167.397,46.849,158.635
C02554=1025.695,-2.538,-95.406,167.394,46.852,158.635
C02555=1025.689,-2.788,-95.391,167.391,46.855,158.635
C02556=1025.683,-3.038,-95.377,167.389,46.857,158.636
C02557=1025.676,-3.287,-95.363,167.386,46.860,158.636
C02558=1025.670,-3.537,-95.349,167.383,46.863,158.636
C02559=1025.664,-3.786,-95.334,167.381,46.865,158.636
C02560=1025.659,-4.036,-95.320,167.378,46.868,158.636
C02561=1025.651,-4.318,-95.304,167.375,46.871,158.636
C02562=1025.645,-4.600,-95.288,167.372,46.875,158.637
C02563=1025.638,-4.881,-95.272,167.369,46.878,158.637
C02564=1025.630,-5.164,-95.257,167.366,46.882,158.637
C02565=1025.624,-5.414,-95.243,167.363,46.885,158.638
C02566=1025.619,-5.663,-95.228,167.360,46.888,158.638
C02567=1025.612,-5.913,-95.214,167.358,46.891,158.638
C02568=1025.606,-6.163,-95.201,167.355,46.894,158.638
C02569=1025.600,-6.412,-95.187,167.353,46.897,158.638
C02570=1025.594,-6.662,-95.172,167.350,46.899,158.639
C02571=1025.588,-6.911,-95.159,167.347,46.903,158.639
C02572=1025.581,-7.161,-95.145,167.345,46.905,158.639
C02573=1025.575,-7.410,-95.131,167.342,46.908,158.639
C02574=1025.569,-7.659,-95.117,167.340,46.912,158.640
C02575=1025.563,-7.909,-95.103,167.336,46.915,158.640
C02576=1025.557,-8.159,-95.090,167.334,46.918,158.640
C02577=1025.550,-8.408,-95.075,167.331,46.921,158.640
C02578=1025.545,-8.658,-95.061,167.329,46.924,158.640
C02579=1025.539,-8.907,-95.047,167.326,46.927,158.641
C02580=1025.532,-9.157,-95.034,167.323,46.930,158.641
C02581=1025.527,-9.407,-95.020,167.320,46.933,158.641
C02582=1025.520,-9.656,-95.006,167.318,46.935,158.641
C02583=1025.514,-9.906,-94.992,167.315,46.938,158.641
C02584=1025.508,-10.155,-94.978,167.312,46.941,158.642
C02585=1025.502,-10.405,-94.965,167.309,46.944,158.642
C02586=1025.496,-10.655,-94.951,167.307,46.947,158.642
C02587=1025.490,-10.904,-94.936,167.304,46.950,158.642
C02588=1025.484,-11.153,-94.923,167.302,46.953,158.642
C02589=1025.478,-11.403,-94.909,167.298,46.956,158.643
C02590=1025.471,-11.652,-94.896,167.296,46.959,158.643
C02591=1025.466,-11.902,-94.882,167.294,46.962,158.643
C02592=1025.460,-12.151,-94.868,167.291,46.965,158.643
C02593=1025.454,-12.402,-94.854,167.288,46.968,158.643
C02594=1025.447,-12.650,-94.840,167.285,46.971,158.644
C02595=1025.442,-12.900,-94.826,167.283,46.974,158.644
C02596=1025.435,-13.150,-94.813,167.280,46.977,158.644
C02597=1025.429,-13.399,-94.799,167.278,46.979,158.644
C02598=1025.423,-13.649,-94.786,167.274,46.983,158.644
C02599=1025.418,-13.898,-94.772,167.272,46.985,158.644
C02600=1025.411,-14.148,-94.758,167.269,46.988,158.645
C02601=1025.405,-14.398,-94.744,167.266,46.991,158.645
C02602=1025.399,-14.647,-94.731,167.263,46.994,158.645
C02603=1025.394,-14.897,-94.717,167.261,46.996,158.645
C02604=1025.387,-15.147,-94.703,167.258,47.000,158.645
C02605=1025.381,-15.396,-94.690,167.255,47.002,158.646
C02606=1025.375,-15.645,-94.676,167.252,47.005,158.646
C02607=1025.370,-15.895,-94.662,167.250,47.008,158.646
C02608=1025.363,-16.145,-94.649,167.247,47.011,158.646
C02609=1025.357,-16.394,-94.636,167.245,47.014,158.646
C02610=1025.350,-16.643,-94.622,167.241,47.017,158.647
C02611=1025.345,-16.893,-94.608,167.239,47.020,158.647
C02612=1025.338,-17.143,-94.595,167.236,47.024,158.647
C02613=1025.332,-17.392,-94.582,167.234,47.027,158.647
C02614=1025.326,-17.642,-94.569,167.231,47.030,158.648
C02615=1025.321,-17.892,-94.555,167.229,47.033,158.648
C02616=1025.314,-18.141,-94.542,167.225,47.036,158.648
C02617=1025.308,-18.391,-94.528,167.222,47.039,158.648
C02618=1025.301,-18.640,-94.515,167.220,47.042,158.648
C02619=1025.296,-18.890,-94.501,167.217,47.045,158.649
C02620=1025.290,-19.139,-94.488,167.214,47.047,158.649
C02621=1025.284,-19.389,-94.475,167.211,47.051,158.649
C02622=1025.277,-19.638,-94.462,167.209,47.053,158.649
C02623=1025.271,-19.888,-94.448,167.206,47.056,158.649
C02624=1025.265,-20.138,-94.434,167.204,47.059,158.650
C02625=1025.255,-20.551,-94.413,167.199,47.064,158.650
C02626=1025.245,-20.965,-94.391,167.194,47.069,158.650
C02627=1025.235,-21.378,-94.369,167.189,47.074,158.650
C02628=1025.225,-21.792,-94.347,167.185,47.079,158.651
C02629=1025.219,-22.042,-94.333,167.183,47.082,158.651
C02630=1025.213,-22.291,-94.320,167.179,47.085,158.651
C02631=1025.207,-22.541,-94.308,167.177,47.088,158.651
C02632=1025.201,-22.790,-94.294,167.174,47.091,158.652
C02633=1025.195,-23.040,-94.280,167.172,47.094,158.652
C02634=1025.189,-23.289,-94.268,167.168,47.097,158.652
C02635=1025.183,-23.539,-94.255,167.165,47.100,158.652
C02636=1025.176,-23.789,-94.241,167.163,47.103,158.652
C02637=1025.171,-24.039,-94.228,167.160,47.106,158.653
C02638=1025.165,-24.288,-94.214,167.158,47.109,158.653
C02639=1025.158,-24.537,-94.201,167.154,47.112,158.653
C02640=1025.152,-24.787,-94.188,167.152,47.115,158.653
C02641=1025.146,-25.037,-94.175,167.149,47.118,158.653
C02642=1025.141,-25.286,-94.162,167.147,47.121,158.654
C02643=1025.135,-25.536,-94.149,167.143,47.124,158.654
C02644=1025.129,-25.785,-94.136,167.141,47.127,158.654
C02645=1025.122,-26.035,-94.122,167.138,47.130,158.654
C02646=1025.117,-26.284,-94.110,167.136,47.132,158.654
C02647=1025.111,-26.534,-94.096,167.133,47.136,158.654
C02648=1025.105,-26.783,-94.083,167.129,47.139,158.655
C02649=1025.099,-27.033,-94.070,167.127,47.142,158.655
C02650=1025.093,-27.282,-94.057,167.124,47.145,158.655
C02651=1025.087,-27.532,-94.044,167.122,47.147,158.655
C02652=1025.081,-27.782,-94.031,167.118,47.151,158.655
C02653=1025.075,-28.031,-94.019,167.116,47.153,158.656
C02654=1025.069,-28.281,-94.005,167.113,47.156,158.656
C02655=1025.063,-28.531,-93.993,167.110,47.160,158.656
C02656=1025.057,-28.780,-93.980,167.108,47.162,158.656
C02657=1025.050,-29.030,-93.967,167.104,47.165,158.656
C02658=1025.045,-29.280,-93.954,167.102,47.169,158.657
C02659=1025.038,-29.529,-93.941,167.099,47.172,158.657
C02660=1025.032,-29.779,-93.929,167.096,47.175,158.657
C02661=1025.026,-30.028,-93.915,167.094,47.178,158.657
C02662=1025.020,-30.278,-93.903,167.091,47.181,158.657
C02663=1025.014,-30.528,-93.890,167.087,47.184,158.658
C02664=1025.007,-30.777,-93.877,167.085,47.187,158.658
C02665=1025.002,-31.027,-93.865,167.082,47.190,158.658
C02666=1024.996,-31.277,-93.852,167.080,47.193,158.658
C02667=1024.989,-31.526,-93.839,167.076,47.196,158.658
C02668=1024.984,-31.776,-93.827,167.073,47.199,158.658
C02669=1024.977,-32.025,-93.813,167.071,47.202,158.659
C02670=1024.971,-32.275,-93.801,167.068,47.205,158.659
C02671=1024.966,-32.525,-93.788,167.066,47.208,158.659
C02672=1024.959,-32.774,-93.775,167.062,47.211,158.659
C02673=1024.953,-33.024,-93.762,167.059,47.215,158.660
C02674=1024.947,-33.274,-93.750,167.057,47.218,158.660
C02675=1024.942,-33.524,-93.737,167.054,47.221,158.660
C02676=1024.935,-33.773,-93.725,167.051,47.224,158.660
C02677=1024.927,-34.139,-93.706,167.047,47.228,158.660
C02678=1024.918,-34.505,-93.687,167.043,47.232,158.661
C02679=1024.909,-34.871,-93.668,167.039,47.237,158.661
C02680=1024.900,-35.237,-93.650,167.034,47.241,158.661
C02681=1024.894,-35.487,-93.638,167.032,47.244,158.661
C02682=1024.888,-35.737,-93.625,167.029,47.247,158.661
C02683=1024.882,-35.986,-93.613,167.026,47.250,158.662
C02684=1024.876,-36.236,-93.599,167.023,47.253,158.662
C02685=1024.869,-36.515,-93.586,167.020,47.257,158.662
C02686=1024.863,-36.795,-93.572,167.017,47.260,158.662
C02687=1024.856,-37.074,-93.557,167.014,47.263,158.662
C02688=1024.850,-37.354,-93.544,167.011,47.267,158.663
C02689=1024.844,-37.604,-93.532,167.008,47.270,158.663
C02690=1024.837,-37.853,-93.519,167.006,47.273,158.663
C02691=1024.831,-38.103,-93.506,167.002,47.276,158.663
C02692=1024.826,-38.353,-93.493,166.999,47.279,158.663
C02693=1024.820,-38.602,-93.481,166.997,47.282,158.664
C02694=1024.814,-38.852,-93.469,166.994,47.285,158.664
C02695=1024.808,-39.102,-93.456,166.990,47.287,158.664
C02696=1024.802,-39.351,-93.444,166.988,47.291,158.664
C02697=1024.796,-39.601,-93.432,166.985,47.294,158.664
C02698=1024.790,-39.851,-93.419,166.982,47.297,158.664
C02699=1024.784,-40.100,-93.407,166.980,47.300,158.665
C02700=1024.778,-40.350,-93.395,166.976,47.303,158.665
C02701=1024.772,-40.600,-93.382,166.973,47.306,158.665
C02702=1024.765,-40.849,-93.370,166.971,47.309,158.665
C02703=1024.760,-41.099,-93.358,166.968,47.312,158.665
C02704=1024.754,-41.348,-93.346,166.965,47.316,158.666
C02705=1024.748,-41.598,-93.334,166.963,47.319,158.666
C02706=1024.742,-41.848,-93.321,166.959,47.322,158.666
C02707=1024.735,-42.097,-93.309,166.956,47.325,158.666
C02708=1024.730,-42.346,-93.297,166.954,47.328,158.666
C02709=1024.724,-42.596,-93.284,166.951,47.331,158.667
C02710=1024.717,-42.846,-93.272,166.948,47.334,158.667
C02711=1024.711,-43.096,-93.260,166.945,47.337,158.667
C02712=1024.705,-43.345,-93.248,166.942,47.340,158.667
C02713=1024.699,-43.595,-93.236,166.939,47.343,158.667
C02714=1024.693,-43.844,-93.223,166.937,47.347,158.668
C02715=1024.688,-44.094,-93.212,166.934,47.350,158.668
C02716=1024.682,-44.344,-93.200,166.931,47.353,158.668
C02717=1024.676,-44.594,-93.187,166.927,47.356,158.668
C02718=1024.669,-44.843,-93.175,166.925,47.359,158.668
C02719=1024.664,-45.092,-93.163,166.922,47.362,158.668
C02720=1024.657,-45.342,-93.151,166.919,47.365,158.669
C02721=1024.651,-45.592,-93.139,166.916,47.368,158.669
C02722=1024.646,-45.842,-93.127,166.913,47.371,158.669
C02723=1024.640,-46.091,-93.115,166.910,47.374,158.669
C02724=1024.634,-46.341,-93.103,166.908,47.377,158.669
C02725=1024.628,-46.590,-93.091,166.905,47.380,158.669
C02726=1024.622,-46.840,-93.078,166.901,47.383,158.670
C02727=1024.616,-47.090,-93.067,166.899,47.386,158.670
C02728=1024.610,-47.339,-93.055,166.896,47.389,158.670
C02729=1024.604,-47.589,-93.042,166.893,47.392,158.670
C02730=1024.598,-47.838,-93.031,166.891,47.395,158.670
C02731=1024.592,-48.088,-93.018,166.887,47.398,158.670
C02732=1024.587,-48.338,-93.006,166.884,47.402,158.671
C02733=1024.581,-48.587,-92.995,166.882,47.404,158.671
C02734=1024.575,-48.837,-92.982,166.879,47.408,158.671
C02735=1024.569,-49.087,-92.971,166.875,47.411,158.671
C02736=1024.563,-49.337,-92.959,166.873,47.414,158.671
C02737=1024.556,-49.586,-92.947,166.870,47.417,158.671
C02738=1024.551,-49.835,-92.935,166.867,47.420,158.672
C02739=1024.546,-50.086,-92.923,166.865,47.423,158.672
C02740=1024.540,-50.335,-92.911,166.861,47.426,158.672
C02741=1024.534,-50.585,-92.899,166.858,47.429,158.672
C02742=1024.527,-50.835,-92.888,166.856,47.432,158.672
C02743=1024.522,-51.084,-92.875,166.853,47.436,158.673
C02744=1024.516,-51.334,-92.864,166.850,47.439,158.673
C02745=1024.510,-51.583,-92.852,166.847,47.442,158.673
C02746=1024.503,-51.833,-92.841,166.843,47.445,158.673
C02747=1024.497,-52.083,-92.829,166.842,47.448,158.673
C02748=1024.492,-52.333,-92.818,166.838,47.452,158.674
C02749=1024.485,-52.612,-92.805,166.835,47.455,158.674
C02750=1024.477,-52.893,-92.791,166.831,47.459,158.674
C02751=1024.471,-53.173,-92.779,166.828,47.463,158.674
C02752=1024.464,-53.453,-92.766,166.825,47.466,158.674
C02753=1024.458,-53.702,-92.755,166.822,47.470,158.675
C02754=1024.451,-53.952,-92.743,166.819,47.473,158.675
C02755=1024.446,-54.201,-92.731,166.816,47.476,158.675
C02756=1024.440,-54.451,-92.720,166.813,47.479,158.675
C02757=1024.433,-54.701,-92.708,166.810,47.483,158.675
C02758=1024.428,-54.951,-92.697,166.807,47.486,158.676
C02759=1024.421,-55.200,-92.685,166.804,47.489,158.676
C02760=1024.416,-55.450,-92.674,166.801,47.492,158.676
C02761=1024.410,-55.700,-92.663,166.799,47.495,158.676
C02762=1024.404,-55.949,-92.651,166.796,47.499,158.676
C02763=1024.397,-56.199,-92.640,166.793,47.502,158.677
C02764=1024.391,-56.448,-92.628,166.789,47.505,158.677
C02765=1024.385,-56.698,-92.617,166.787,47.508,158.677
C02766=1024.380,-56.948,-92.606,166.784,47.511,158.677
C02767=1024.374,-57.197,-92.594,166.781,47.515,158.677
C02768=1024.367,-57.447,-92.583,166.778,47.518,158.677
C02769=1024.362,-57.697,-92.572,166.775,47.521,158.678
C02770=1024.355,-57.946,-92.560,166.772,47.524,158.678
C02771=1024.349,-58.196,-92.549,166.769,47.527,158.678
C02772=1024.344,-58.446,-92.537,166.766,47.530,158.678
C02773=1024.338,-58.696,-92.526,166.763,47.534,158.678
C02774=1024.331,-58.945,-92.514,166.760,47.537,158.678
C02775=1024.326,-59.195,-92.503,166.758,47.540,158.679
C02776=1024.320,-59.444,-92.493,166.754,47.543,158.679
C02777=1024.314,-59.694,-92.480,166.751,47.546,158.679
C02778=1024.308,-59.944,-92.469,166.748,47.549,158.679
C02779=1024.302,-60.194,-92.458,166.746,47.553,158.680
C02780=1024.296,-60.443,-92.447,166.743,47.556,158.680
C02781=1024.290,-60.693,-92.436,166.740,47.559,158.680
C02782=1024.284,-60.942,-92.424,166.736,47.562,158.680
C02783=1024.278,-61.192,-92.413,166.733,47.566,158.680
C02784=1024.273,-61.442,-92.402,166.731,47.568,158.680
C02785=1024.267,-61.692,-92.391,166.728,47.572,158.680
C02786=1024.261,-61.941,-92.380,166.725,47.575,158.681
C02787=1024.254,-62.191,-92.368,166.722,47.579,158.681
C02788=1024.249,-62.441,-92.357,166.718,47.582,158.681
C02789=1024.243,-62.690,-92.346,166.716,47.585,158.681
C02790=1024.237,-62.941,-92.334,166.713,47.588,158.681
C02791=1024.231,-63.190,-92.323,166.710,47.591,158.681
C02792=1024.226,-63.439,-92.312,166.707,47.594,158.682
C02793=1024.220,-63.689,-92.302,166.704,47.597,158.682
///RCONF 1,0,0,1,0,0,0,0,0,0,0,0,0,0,0,0,0,0,0,0,0,0,0,0
C02794=1024.213,-63.939,-92.290,166.701,47.600,158.682
C02795=1024.208,-64.188,-92.279,166.698,47.603,158.682
C02796=1024.202,-64.438,-92.268,166.695,47.607,158.682
C02797=1024.196,-64.688,-92.256,166.692,47.610,158.682
C02798=1024.191,-64.938,-92.245,166.690,47.613,158.683
C02799=1024.185,-65.187,-92.234,166.686,47.616,158.683
C02800=1024.178,-65.437,-92.223,166.683,47.619,158.683
C02801=1024.173,-65.687,-92.212,166.680,47.622,158.683
C02802=1024.167,-65.936,-92.201,166.678,47.625,158.683
C02803=1024.161,-66.186,-92.190,166.675,47.628,158.683
C02804=1024.155,-66.436,-92.179,166.671,47.632,158.684
C02805=1024.150,-66.686,-92.168,166.668,47.635,158.684
C02806=1024.144,-66.935,-92.157,166.666,47.638,158.684
C02807=1024.138,-67.185,-92.146,166.663,47.641,158.684
C02808=1024.132,-67.435,-92.135,166.660,47.645,158.684
C02809=1024.126,-67.684,-92.124,166.657,47.648,158.684
C02810=1024.121,-67.934,-92.113,166.653,47.651,158.685
C02811=1024.115,-68.183,-92.102,166.651,47.654,158.685
C02812=1024.109,-68.433,-92.091,166.648,47.657,158.685
C02813=1024.103,-68.714,-92.078,166.645,47.660,158.685
C02814=1024.096,-68.996,-92.066,166.641,47.664,158.685
C02815=1024.089,-69.277,-92.054,166.638,47.667,158.685
C02816=1024.083,-69.558,-92.041,166.634,47.670,158.686
C02817=1024.077,-69.808,-92.030,166.631,47.674,158.686
C02818=1024.072,-70.057,-92.019,166.628,47.677,158.686
C02819=1024.066,-70.307,-92.008,166.626,47.680,158.686
C02820=1024.060,-70.557,-91.998,166.623,47.684,158.686
C02821=1024.055,-70.806,-91.987,166.620,47.687,158.686
C02822=1024.048,-71.056,-91.976,166.616,47.690,158.687
C02823=1024.043,-71.306,-91.964,166.614,47.693,158.687
C02824=1024.038,-71.556,-91.953,166.611,47.696,158.687
C02825=1024.032,-71.805,-91.943,166.608,47.699,158.687
C02826=1024.026,-72.055,-91.932,166.605,47.702,158.687
C02827=1024.020,-72.304,-91.921,166.601,47.705,158.687
C02828=1024.015,-72.554,-91.911,166.599,47.708,158.687
C02829=1024.009,-72.804,-91.900,166.596,47.711,158.688
C02830=1024.003,-73.054,-91.889,166.593,47.715,158.688
C02831=1023.997,-73.303,-91.878,166.590,47.718,158.688
C02832=1023.991,-73.553,-91.867,166.587,47.721,158.688
C02833=1023.987,-73.803,-91.856,166.584,47.724,158.688
C02834=1023.981,-74.053,-91.845,166.581,47.727,158.688
C02835=1023.975,-74.302,-91.834,166.578,47.730,158.688
C02836=1023.969,-74.552,-91.823,166.576,47.733,158.689
C02837=1023.963,-74.802,-91.814,166.572,47.736,158.689
C02838=1023.958,-75.051,-91.803,166.569,47.739,158.689
C02839=1023.952,-75.301,-91.792,166.566,47.742,158.689
C02840=1023.946,-75.551,-91.782,166.563,47.746,158.689
C02841=1023.940,-75.801,-91.771,166.560,47.749,158.689
C02842=1023.934,-76.051,-91.761,166.557,47.753,158.690
C02843=1023.928,-76.300,-91.750,166.554,47.755,158.690
C02844=1023.922,-76.550,-91.739,166.551,47.759,158.690
C02845=1023.917,-76.800,-91.729,166.548,47.762,158.690
C02846=1023.911,-77.049,-91.718,166.545,47.766,158.690
C02847=1023.905,-77.299,-91.709,166.542,47.769,158.690
C02848=1023.899,-77.548,-91.698,166.539,47.772,158.691
C02849=1023.894,-77.798,-91.687,166.537,47.775,158.691
C02850=1023.888,-78.048,-91.677,166.533,47.778,158.691
C02851=1023.882,-78.298,-91.666,166.530,47.781,158.691
C02852=1023.876,-78.547,-91.656,166.527,47.784,158.691
C02853=1023.870,-78.797,-91.646,166.524,47.788,158.691
C02854=1023.865,-79.047,-91.635,166.521,47.791,158.692
C02855=1023.859,-79.296,-91.624,166.518,47.795,158.692
C02856=1023.853,-79.546,-91.615,166.515,47.797,158.692
C02857=1023.847,-79.796,-91.604,166.512,47.801,158.692
C02858=1023.842,-80.046,-91.594,166.509,47.804,158.692
C02859=1023.836,-80.295,-91.583,166.506,47.808,158.692
C02860=1023.830,-80.545,-91.573,166.503,47.811,158.693
C02861=1023.825,-80.795,-91.563,166.500,47.814,158.693
C02862=1023.818,-81.044,-91.553,166.496,47.817,158.693
C02863=1023.813,-81.295,-91.543,166.494,47.821,158.693
C02864=1023.807,-81.544,-91.533,166.490,47.824,158.693
C02865=1023.801,-81.794,-91.522,166.488,47.827,158.693
C02866=1023.795,-82.044,-91.513,166.485,47.831,158.694
C02867=1023.789,-82.294,-91.503,166.482,47.834,158.694
C02868=1023.783,-82.543,-91.492,166.479,47.837,158.694
C02869=1023.778,-82.792,-91.483,166.476,47.841,158.694
C02870=1023.772,-83.042,-91.473,166.473,47.844,158.694
C02871=1023.766,-83.292,-91.462,166.470,47.847,158.694
C02872=1023.760,-83.541,-91.453,166.467,47.851,158.695
C02873=1023.754,-83.792,-91.442,166.463,47.855,158.695
C02874=1023.748,-84.041,-91.433,166.460,47.858,158.695
C02875=1023.742,-84.291,-91.422,166.457,47.861,158.695
C02876=1023.737,-84.541,-91.412,166.454,47.865,158.695
C02877=1023.730,-84.825,-91.401,166.451,47.868,158.696
C02878=1023.724,-85.107,-91.390,166.448,47.872,158.696
C02879=1023.717,-85.391,-91.378,166.444,47.876,158.696
C02880=1023.711,-85.674,-91.367,166.441,47.880,158.696
C02881=1023.704,-85.924,-91.357,166.438,47.883,158.696
C02882=1023.699,-86.174,-91.347,166.435,47.886,158.697
C02883=1023.692,-86.423,-91.337,166.432,47.889,158.697
C02884=1023.688,-86.673,-91.327,166.429,47.893,158.697
C02885=1023.681,-86.923,-91.318,166.425,47.896,158.697
C02886=1023.676,-87.173,-91.307,166.422,47.900,158.697
C02887=1023.670,-87.422,-91.297,166.419,47.903,158.697
C02888=1023.664,-87.672,-91.287,166.416,47.907,158.698
C02889=1023.659,-87.921,-91.278,166.413,47.910,158.698
C02890=1023.653,-88.171,-91.268,166.411,47.913,158.698
C02891=1023.647,-88.421,-91.258,166.408,47.916,158.698
C02892=1023.642,-88.671,-91.248,166.405,47.920,158.698
C02893=1023.635,-88.921,-91.238,166.401,47.923,158.698
C02894=1023.631,-89.170,-91.229,166.398,47.926,158.698
C02895=1023.624,-89.420,-91.219,166.395,47.929,158.699
C02896=1023.619,-89.670,-91.208,166.392,47.932,158.699
C02897=1023.612,-89.919,-91.199,166.389,47.936,158.699
C02898=1023.607,-90.170,-91.188,166.386,47.940,158.699
C02899=1023.601,-90.419,-91.179,166.382,47.943,158.699
C02900=1023.596,-90.669,-91.169,166.380,47.946,158.699
C02901=1023.590,-90.919,-91.159,166.377,47.949,158.700
C02902=1023.585,-91.168,-91.150,166.374,47.953,158.700
C02903=1023.579,-91.418,-91.140,166.371,47.956,158.700
C02904=1023.573,-91.668,-91.130,166.368,47.959,158.700
C02905=1023.567,-91.918,-91.120,166.365,47.962,158.700
C02906=1023.562,-92.167,-91.111,166.362,47.966,158.700
C02907=1023.556,-92.417,-91.101,166.358,47.969,158.701
C02908=1023.550,-92.667,-91.091,166.355,47.972,158.701
C02909=1023.545,-92.916,-91.082,166.353,47.975,158.701
C02910=1023.539,-93.166,-91.072,166.350,47.979,158.701
C02911=1023.534,-93.416,-91.062,166.347,47.982,158.701
C02912=1023.528,-93.665,-91.053,166.344,47.986,158.701
C02913=1023.523,-93.915,-91.043,166.341,47.989,158.702
C02914=1023.516,-94.165,-91.033,166.337,47.992,158.702
C02915=1023.512,-94.415,-91.024,166.334,47.995,158.702
C02916=1023.506,-94.665,-91.014,166.331,47.998,158.702
C02917=1023.500,-94.915,-91.005,166.328,48.002,158.702
C02918=1023.495,-95.164,-90.995,166.326,48.005,158.702
C02919=1023.489,-95.414,-90.985,166.323,48.008,158.702
C02920=1023.483,-95.664,-90.975,166.320,48.012,158.703
C02921=1023.478,-95.913,-90.966,166.316,48.015,158.703
C02922=1023.472,-96.163,-90.956,166.313,48.018,158.703
C02923=1023.467,-96.412,-90.947,166.310,48.022,158.703
C02924=1023.461,-96.663,-90.937,166.307,48.025,158.703
C02925=1023.455,-96.913,-90.928,166.304,48.028,158.703
C02926=1023.450,-97.162,-90.918,166.302,48.031,158.703
C02927=1023.444,-97.412,-90.908,166.298,48.034,158.704
C02928=1023.439,-97.661,-90.899,166.295,48.037,158.704
C02929=1023.434,-97.912,-90.890,166.292,48.041,158.704
C02930=1023.427,-98.162,-90.880,166.289,48.045,158.704
C02931=1023.422,-98.411,-90.871,166.286,48.048,158.704
C02932=1023.416,-98.660,-90.861,166.283,48.052,158.704
C02933=1023.410,-98.910,-90.853,166.280,48.055,158.705
C02934=1023.405,-99.160,-90.843,166.277,48.058,158.705
C02935=1023.399,-99.410,-90.833,166.274,48.062,158.705
C02936=1023.394,-99.660,-90.825,166.271,48.065,158.705
C02937=1023.387,-99.910,-90.815,166.267,48.068,158.705
C02938=1023.382,-100.159,-90.806,166.264,48.072,158.705
C02939=1023.376,-100.409,-90.797,166.261,48.075,158.706
C02940=1023.371,-100.659,-90.787,166.258,48.079,158.706
C02941=1023.364,-100.944,-90.777,166.255,48.083,158.706
C02942=1023.358,-101.229,-90.766,166.251,48.087,158.706
C02943=1023.351,-101.515,-90.756,166.248,48.091,158.706
C02944=1023.345,-101.801,-90.746,166.244,48.094,158.706
C02945=1023.339,-102.050,-90.736,166.241,48.098,158.707
C02946=1023.333,-102.300,-90.728,166.238,48.101,158.707
C02947=1023.328,-102.549,-90.718,166.235,48.104,158.707
C02948=1023.322,-102.800,-90.708,166.232,48.108,158.707
C02949=1023.317,-103.049,-90.700,166.230,48.111,158.707
C02950=1023.311,-103.299,-90.690,166.227,48.114,158.707
C02951=1023.306,-103.549,-90.682,166.223,48.118,158.708
C02952=1023.300,-103.799,-90.672,166.220,48.121,158.708
C02953=1023.294,-104.048,-90.664,166.217,48.125,158.708
C02954=1023.288,-104.298,-90.654,166.214,48.128,158.708
C02955=1023.284,-104.548,-90.645,166.211,48.132,158.708
C02956=1023.277,-104.798,-90.635,166.208,48.135,158.708
C02957=1023.272,-105.048,-90.627,166.205,48.138,158.709
C02958=1023.267,-105.297,-90.618,166.202,48.142,158.709
C02959=1023.261,-105.547,-90.609,166.199,48.145,158.709
C02960=1023.255,-105.797,-90.600,166.195,48.149,158.709
C02961=1023.249,-106.047,-90.591,166.192,48.152,158.709
C02962=1023.244,-106.296,-90.582,166.189,48.156,158.709
C02963=1023.238,-106.545,-90.573,166.186,48.159,158.710
C02964=1023.233,-106.796,-90.564,166.183,48.162,158.710
C02965=1023.228,-107.046,-90.555,166.180,48.166,158.710
C02966=1023.222,-107.296,-90.546,166.177,48.169,158.710
C02967=1023.217,-107.545,-90.537,166.174,48.172,158.710
C02968=1023.211,-107.795,-90.528,166.172,48.176,158.710
C02969=1023.205,-108.045,-90.519,166.169,48.179,158.711
C02970=1023.200,-108.295,-90.511,166.165,48.182,158.711
C02971=1023.194,-108.545,-90.502,166.163,48.186,158.711
C02972=1023.188,-108.794,-90.493,166.159,48.190,158.711
C02973=1023.183,-109.044,-90.484,166.157,48.193,158.711
C02974=1023.177,-109.294,-90.476,166.153,48.197,158.711
C02975=1023.171,-109.543,-90.467,166.150,48.200,158.712
C02976=1023.166,-109.793,-90.458,166.147,48.204,158.712
C02977=1023.160,-110.043,-90.449,166.144,48.207,158.712
C02978=1023.155,-110.293,-90.441,166.141,48.210,158.712
C02979=1023.149,-110.543,-90.432,166.138,48.214,158.712
C02980=1023.143,-110.792,-90.423,166.135,48.217,158.712
C02981=1023.138,-111.042,-90.414,166.132,48.221,158.713
C02982=1023.133,-111.292,-90.406,166.129,48.224,158.713
C02983=1023.127,-111.542,-90.397,166.125,48.228,158.713
C02984=1023.122,-111.792,-90.388,166.123,48.232,158.713
C02985=1023.116,-112.041,-90.379,166.119,48.235,158.713
C02986=1023.111,-112.291,-90.371,166.116,48.238,158.713
C02987=1023.105,-112.541,-90.362,166.113,48.242,158.714
C02988=1023.099,-112.791,-90.354,166.110,48.245,158.714
C02989=1023.094,-113.040,-90.346,166.107,48.248,158.714
C02990=1023.088,-113.290,-90.337,166.104,48.252,158.714
C02991=1023.082,-113.540,-90.327,166.101,48.255,158.714
C02992=1023.077,-113.790,-90.319,166.098,48.259,158.714
C02993=1023.072,-114.039,-90.311,166.095,48.263,158.715
C02994=1023.066,-114.289,-90.302,166.092,48.266,158.715
C02995=1023.060,-114.539,-90.293,166.088,48.269,158.715
C02996=1023.055,-114.789,-90.285,166.086,48.273,158.715
C02997=1023.049,-115.039,-90.277,166.082,48.276,158.715
C02998=1023.044,-115.288,-90.268,166.079,48.280,158.715
C02999=1023.038,-115.539,-90.259,166.076,48.283,158.715
C03000=1023.033,-115.788,-90.251,166.073,48.287,158.716
C03001=1023.028,-116.038,-90.243,166.070,48.290,158.716
C03002=1023.022,-116.288,-90.235,166.067,48.294,158.716
C03003=1023.016,-116.537,-90.226,166.064,48.298,158.716
C03004=1023.010,-116.788,-90.217,166.061,48.301,158.716
C03005=1023.004,-117.073,-90.208,166.058,48.305,158.717
C03006=1022.998,-117.357,-90.198,166.054,48.309,158.717
C03007=1022.992,-117.642,-90.189,166.051,48.313,158.717
C03008=1022.985,-117.928,-90.179,166.047,48.317,158.717
C03009=1022.980,-118.178,-90.171,166.044,48.320,158.717
C03010=1022.975,-118.428,-90.162,166.041,48.323,158.717
C03011=1022.969,-118.678,-90.154,166.038,48.327,158.718
C03012=1022.963,-118.927,-90.146,166.035,48.331,158.718
C03013=1022.958,-119.177,-90.138,166.032,48.335,158.718
C03014=1022.953,-119.426,-90.129,166.029,48.338,158.718
C03015=1022.947,-119.677,-90.120,166.026,48.342,158.718
C03016=1022.941,-119.926,-90.112,166.023,48.345,158.718
C03017=1022.936,-120.177,-90.105,166.020,48.348,158.719
C03018=1022.931,-120.426,-90.096,166.017,48.352,158.719
C03019=1022.925,-120.676,-90.088,166.013,48.355,158.719
C03020=1022.919,-120.925,-90.080,166.011,48.359,158.719
C03021=1022.914,-121.175,-90.071,166.007,48.362,158.719
C03022=1022.909,-121.426,-90.064,166.004,48.366,158.719
C03023=1022.903,-121.675,-90.056,166.001,48.370,158.720
C03024=1022.898,-121.925,-90.047,165.998,48.373,158.720
C03025=1022.893,-122.174,-90.039,165.995,48.377,158.720
C03026=1022.887,-122.424,-90.031,165.992,48.380,158.720
C03027=1022.881,-122.675,-90.023,165.989,48.383,158.720
C03028=1022.876,-122.925,-90.014,165.986,48.387,158.720
C03029=1022.870,-123.174,-90.006,165.983,48.390,158.720
C03030=1022.865,-123.424,-89.998,165.980,48.394,158.721
C03031=1022.860,-123.674,-89.990,165.978,48.397,158.721
C03032=1022.854,-123.923,-89.982,165.975,48.401,158.721
C03033=1022.848,-124.173,-89.974,165.972,48.404,158.721
C03034=1022.843,-124.423,-89.966,165.968,48.408,158.721
C03035=1022.837,-124.673,-89.958,165.966,48.412,158.722
C03036=1022.832,-124.923,-89.949,165.962,48.415,158.722
C03037=1022.826,-125.173,-89.942,165.960,48.419,158.722
C03038=1022.821,-125.422,-89.934,165.956,48.422,158.722
C03039=1022.815,-125.672,-89.927,165.953,48.426,158.722
C03040=1022.810,-125.922,-89.918,165.950,48.429,158.722
C03041=1022.805,-126.172,-89.910,165.947,48.433,158.723
C03042=1022.799,-126.422,-89.902,165.944,48.436,158.723
C03043=1022.794,-126.671,-89.894,165.941,48.440,158.723
C03044=1022.788,-126.922,-89.887,165.938,48.444,158.723
C03045=1022.783,-127.171,-89.878,165.935,48.448,158.723
C03046=1022.777,-127.421,-89.870,165.932,48.451,158.723
C03047=1022.773,-127.670,-89.863,165.929,48.454,158.724
C03048=1022.767,-127.920,-89.855,165.926,48.458,158.724
C03049=1022.761,-128.169,-89.847,165.923,48.461,158.724
C03050=1022.757,-128.419,-89.838,165.920,48.464,158.724
C03051=1022.753,-128.669,-89.829,165.917,48.466,158.724
C03052=1022.749,-128.918,-89.819,165.914,48.468,158.724
C03053=1022.746,-129.168,-89.809,165.911,48.469,158.724
///RCONF 1,0,0,0,0,0,0,0,0,0,0,0,0,0,0,0,0,0,0,0,0,0,0,0
C03054=1022.744,-129.418,-89.798,165.909,48.471,158.723
C03055=1022.741,-129.668,-89.785,165.906,48.470,158.723
C03056=1022.739,-129.917,-89.774,165.904,48.470,158.723
C03057=1022.739,-130.167,-89.761,165.901,48.469,158.722
C03058=1022.738,-130.417,-89.748,165.899,48.468,158.722
C03059=1022.738,-130.666,-89.733,165.897,48.466,158.721
C03060=1022.738,-130.916,-89.719,165.895,48.464,158.721
C03061=1022.739,-131.166,-89.703,165.893,48.462,158.720
C03062=1022.740,-131.416,-89.688,165.891,48.458,158.719
C03063=1022.742,-131.666,-89.672,165.889,48.455,158.718
C03064=1022.745,-131.916,-89.654,165.888,48.450,158.717
C03065=1022.748,-132.165,-89.637,165.886,48.445,158.716
C03066=1022.751,-132.415,-89.619,165.885,48.440,158.715
C03067=1022.755,-132.665,-89.601,165.882,48.435,158.714
C03068=1022.760,-132.915,-89.581,165.881,48.428,158.712
C03069=1022.469,-132.940,-89.926,165.834,48.721,158.755
C03070=1022.465,-132.691,-89.945,165.835,48.727,158.756
C03071=1022.461,-132.442,-89.964,165.837,48.733,158.758
C03072=1022.458,-132.191,-89.982,165.839,48.738,158.759
C03073=1022.455,-131.941,-89.999,165.840,48.743,158.760
C03074=1022.452,-131.692,-90.016,165.842,48.747,158.761
C03075=1022.451,-131.442,-90.033,165.843,48.751,158.761
C03076=1022.449,-131.193,-90.048,165.846,48.754,158.762
C03077=1022.448,-130.943,-90.064,165.848,48.757,158.763
C03078=1022.448,-130.692,-90.078,165.850,48.759,158.764
C03079=1022.448,-130.443,-90.092,165.852,48.761,158.764
C03080=1022.449,-130.193,-90.106,165.854,48.762,158.765
C03081=1022.450,-129.944,-90.119,165.857,48.763,158.765
C03082=1022.451,-129.693,-90.131,165.859,48.763,158.766
C03083=1022.454,-129.444,-90.143,165.861,48.763,158.766
C03084=1022.456,-129.194,-90.154,165.865,48.762,158.766
C03085=1022.460,-128.945,-90.164,165.867,48.761,158.767
C03086=1022.462,-128.695,-90.174,165.870,48.759,158.767
C03087=1022.467,-128.445,-90.183,165.873,48.757,158.767
C03088=1022.471,-128.195,-90.192,165.875,48.754,158.766
C03089=1022.477,-127.946,-90.200,165.878,48.751,158.766
C03090=1022.482,-127.696,-90.208,165.881,48.747,158.766
C03091=1022.488,-127.446,-90.216,165.884,48.743,158.766
C03092=1022.493,-127.197,-90.224,165.887,48.739,158.766
C03093=1022.498,-126.948,-90.232,165.890,48.736,158.766
C03094=1022.503,-126.698,-90.239,165.894,48.732,158.766
C03095=1022.509,-126.448,-90.248,165.897,48.729,158.765
C03096=1022.514,-126.198,-90.255,165.900,48.725,158.765
C03097=1022.520,-125.948,-90.264,165.903,48.721,158.765
C03098=1022.525,-125.698,-90.271,165.906,48.717,158.765
C03099=1022.531,-125.448,-90.279,165.909,48.714,158.765
C03100=1022.536,-125.198,-90.286,165.912,48.710,158.765
C03101=1022.542,-124.949,-90.295,165.915,48.707,158.764
C03102=1022.548,-124.699,-90.303,165.918,48.703,158.764
C03103=1022.553,-124.449,-90.310,165.921,48.700,158.764
C03104=1022.558,-124.199,-90.319,165.924,48.696,158.764
C03105=1022.564,-123.950,-90.327,165.927,48.692,158.764
C03106=1022.569,-123.699,-90.335,165.930,48.688,158.763
C03107=1022.574,-123.450,-90.343,165.933,48.685,158.763
C03108=1022.580,-123.200,-90.351,165.936,48.681,158.763
C03109=1022.585,-122.950,-90.359,165.939,48.678,158.763
C03110=1022.590,-122.700,-90.367,165.942,48.674,158.763
C03111=1022.596,-122.451,-90.375,165.945,48.671,158.763
C03112=1022.602,-122.201,-90.384,165.948,48.667,158.762
C03113=1022.606,-121.951,-90.391,165.951,48.664,158.762
C03114=1022.612,-121.701,-90.399,165.954,48.660,158.762
C03115=1022.618,-121.452,-90.408,165.957,48.656,158.762
C03116=1022.624,-121.201,-90.417,165.960,48.653,158.762
C03117=1022.629,-120.951,-90.424,165.963,48.649,158.762
C03118=1022.635,-120.702,-90.432,165.966,48.646,158.762
C03119=1022.640,-120.452,-90.441,165.969,48.642,158.761
C03120=1022.645,-120.202,-90.449,165.972,48.639,158.761
C03121=1022.651,-119.953,-90.457,165.975,48.635,158.761
C03122=1022.656,-119.702,-90.465,165.978,48.631,158.761
C03123=1022.661,-119.453,-90.473,165.981,48.628,158.761
C03124=1022.667,-119.203,-90.482,165.985,48.624,158.761
C03125=1022.673,-118.954,-90.490,165.987,48.620,158.760
C03126=1022.678,-118.704,-90.498,165.991,48.617,158.760
C03127=1022.684,-118.453,-90.507,165.993,48.613,158.760
C03128=1022.690,-118.204,-90.515,165.998,48.610,158.760
C03129=1022.695,-117.954,-90.524,166.000,48.606,158.760
C03130=1022.701,-117.669,-90.532,166.004,48.602,158.760
C03131=1022.707,-117.384,-90.542,166.008,48.598,158.759
C03132=1022.713,-117.099,-90.551,166.010,48.594,158.759
C03133=1022.720,-116.813,-90.561,166.014,48.590,158.759
C03134=1022.726,-116.564,-90.570,166.017,48.586,158.759
C03135=1022.731,-116.314,-90.578,166.020,48.583,158.759
C03136=1022.736,-116.064,-90.587,166.023,48.579,158.758
C03137=1022.741,-115.815,-90.595,166.026,48.576,158.758
C03138=1022.747,-115.565,-90.603,166.029,48.572,158.758
C03139=1022.753,-115.315,-90.612,166.032,48.568,158.758
C03140=1022.758,-115.065,-90.620,166.035,48.564,158.758
C03141=1022.764,-114.815,-90.629,166.038,48.561,158.758
C03142=1022.769,-114.566,-90.637,166.042,48.558,158.757
C03143=1022.775,-114.316,-90.645,166.044,48.554,158.757
C03144=1022.781,-114.066,-90.654,166.048,48.551,158.757
C03145=1022.786,-113.816,-90.663,166.050,48.547,158.757
C03146=1022.791,-113.566,-90.671,166.054,48.544,158.757
C03147=1022.797,-113.317,-90.680,166.057,48.540,158.757
C03148=1022.803,-113.066,-90.689,166.060,48.536,158.756
C03149=1022.808,-112.817,-90.697,166.063,48.533,158.756
C03150=1022.813,-112.567,-90.706,166.066,48.529,158.756
C03151=1022.819,-112.318,-90.715,166.069,48.526,158.756
C03152=1022.824,-112.067,-90.724,166.072,48.522,158.756
C03153=1022.830,-111.818,-90.732,166.075,48.519,158.756
C03154=1022.835,-111.568,-90.740,166.078,48.516,158.755
C03155=1022.841,-111.318,-90.748,166.081,48.512,158.755
C03156=1022.847,-111.068,-90.757,166.084,48.508,158.755
C03157=1022.852,-110.819,-90.766,166.087,48.504,158.755
C03158=1022.858,-110.569,-90.775,166.090,48.501,158.755
C03159=1022.864,-110.319,-90.784,166.093,48.497,158.754
C03160=1022.869,-110.069,-90.792,166.096,48.494,158.754
C03161=1022.874,-109.819,-90.801,166.099,48.491,158.754
C03162=1022.880,-109.570,-90.810,166.102,48.487,158.754
C03163=1022.886,-109.320,-90.819,166.105,48.484,158.754
C03164=1022.891,-109.070,-90.827,166.108,48.480,158.754
C03165=1022.896,-108.820,-90.836,166.111,48.476,158.754
C03166=1022.902,-108.571,-90.845,166.115,48.472,158.753
C03167=1022.908,-108.321,-90.854,166.119,48.469,158.753
C03168=1022.913,-108.070,-90.863,166.121,48.465,158.753
C03169=1022.919,-107.821,-90.871,166.125,48.462,158.753
C03170=1022.924,-107.572,-90.880,166.128,48.459,158.753
C03171=1022.930,-107.321,-90.889,166.131,48.455,158.753
C03172=1022.935,-107.072,-90.898,166.134,48.451,158.752
C03173=1022.941,-106.822,-90.907,166.137,48.448,158.752
C03174=1022.947,-106.572,-90.916,166.140,48.444,158.752
C03175=1022.952,-106.323,-90.925,166.143,48.441,158.752
C03176=1022.958,-106.073,-90.934,166.146,48.437,158.752
C03177=1022.963,-105.823,-90.942,166.149,48.434,158.752
C03178=1022.969,-105.574,-90.951,166.152,48.431,158.751
C03179=1022.975,-105.323,-90.960,166.155,48.427,158.751
C03180=1022.980,-105.074,-90.970,166.157,48.424,158.751
C03181=1022.986,-104.823,-90.979,166.160,48.421,158.751
C03182=1022.991,-104.574,-90.987,166.163,48.417,158.751
C03183=1022.996,-104.325,-90.997,166.167,48.413,158.751
C03184=1023.002,-104.074,-91.006,166.170,48.410,158.750
C03185=1023.008,-103.825,-91.015,166.173,48.406,158.750
C03186=1023.014,-103.575,-91.024,166.176,48.403,158.750
C03187=1023.019,-103.326,-91.033,166.179,48.399,158.750
C03188=1023.024,-103.075,-91.042,166.182,48.396,158.750
C03189=1023.030,-102.826,-91.051,166.185,48.393,158.750
C03190=1023.036,-102.575,-91.060,166.188,48.389,158.749
C03191=1023.041,-102.326,-91.069,166.191,48.385,158.749
C03192=1023.047,-102.076,-91.078,166.194,48.382,158.749
C03193=1023.053,-101.827,-91.088,166.197,48.378,158.749
C03194=1023.059,-101.541,-91.098,166.201,48.374,158.749
C03195=1023.066,-101.256,-91.109,166.204,48.371,158.749
C03196=1023.072,-100.971,-91.119,166.208,48.367,158.748
C03197=1023.078,-100.685,-91.130,166.212,48.362,158.748
C03198=1023.084,-100.435,-91.139,166.215,48.359,158.748
C03199=1023.090,-100.186,-91.148,166.218,48.355,158.748
C03200=1023.095,-99.936,-91.157,166.221,48.352,158.748
C03201=1023.101,-99.686,-91.166,166.224,48.348,158.747
C03202=1023.107,-99.437,-91.176,166.227,48.345,158.747
C03203=1023.112,-99.187,-91.185,166.230,48.341,158.747
C03204=1023.118,-98.937,-91.194,166.233,48.338,158.747
C03205=1023.124,-98.687,-91.204,166.237,48.335,158.747
C03206=1023.129,-98.437,-91.212,166.239,48.331,158.747
C03207=1023.135,-98.188,-91.222,166.243,48.327,158.747
C03208=1023.140,-97.938,-91.232,166.245,48.324,158.746
C03209=1023.146,-97.688,-91.241,166.249,48.320,158.746
C03210=1023.152,-97.439,-91.250,166.252,48.317,158.746
C03211=1023.157,-97.188,-91.260,166.254,48.314,158.746
C03212=1023.163,-96.939,-91.270,166.257,48.310,158.746
C03213=1023.169,-96.690,-91.279,166.260,48.307,158.745
C03214=1023.174,-96.439,-91.288,166.263,48.304,158.745
C03215=1023.180,-96.190,-91.297,166.266,48.301,158.745
C03216=1023.185,-95.940,-91.308,166.269,48.297,158.745
C03217=1023.191,-95.691,-91.317,166.272,48.293,158.745
C03218=1023.196,-95.440,-91.327,166.276,48.290,158.745
C03219=1023.202,-95.191,-91.336,166.279,48.287,158.745
C03220=1023.207,-94.941,-91.346,166.282,48.284,158.745
C03221=1023.213,-94.691,-91.355,166.285,48.280,158.744
C03222=1023.219,-94.441,-91.365,166.288,48.277,158.744
C03223=1023.224,-94.192,-91.374,166.291,48.273,158.744
C03224=1023.230,-93.942,-91.384,166.293,48.271,158.744
C03225=1023.235,-93.692,-91.394,166.296,48.267,158.744
C03226=1023.241,-93.443,-91.403,166.299,48.263,158.743
C03227=1023.246,-93.193,-91.414,166.303,48.260,158.743
C03228=1023.252,-92.943,-91.423,166.306,48.257,158.743
C03229=1023.258,-92.693,-91.433,166.309,48.253,158.743
C03230=1023.264,-92.444,-91.442,166.312,48.250,158.743
C03231=1023.269,-92.194,-91.452,166.315,48.247,158.743
C03232=1023.275,-91.944,-91.462,166.318,48.243,158.742
C03233=1023.280,-91.694,-91.472,166.321,48.240,158.742
C03234=1023.286,-91.444,-91.482,166.324,48.236,158.742
C03235=1023.292,-91.195,-91.491,166.328,48.233,158.742
C03236=1023.297,-90.945,-91.501,166.330,48.229,158.742
C03237=1023.303,-90.695,-91.511,166.334,48.226,158.742
C03238=1023.308,-90.446,-91.520,166.337,48.223,158.742
C03239=1023.314,-90.196,-91.530,166.340,48.219,158.741
C03240=1023.320,-89.946,-91.540,166.342,48.216,158.741
C03241=1023.326,-89.696,-91.550,166.345,48.213,158.741
C03242=1023.331,-89.447,-91.559,166.348,48.210,158.741
C03243=1023.337,-89.197,-91.569,166.351,48.206,158.741
C03244=1023.343,-88.947,-91.579,166.354,48.202,158.741
C03245=1023.349,-88.697,-91.589,166.357,48.199,158.740
C03246=1023.354,-88.448,-91.598,166.360,48.195,158.740
C03247=1023.360,-88.198,-91.608,166.363,48.192,158.740
C03248=1023.365,-87.948,-91.618,166.367,48.189,158.740
C03249=1023.371,-87.698,-91.628,166.370,48.185,158.740
C03250=1023.377,-87.449,-91.639,166.373,48.182,158.740
C03251=1023.383,-87.199,-91.648,166.376,48.179,158.739
C03252=1023.388,-86.949,-91.658,166.379,48.175,158.739
C03253=1023.394,-86.700,-91.668,166.382,48.172,158.739
C03254=1023.400,-86.449,-91.678,166.385,48.168,158.739
C03255=1023.406,-86.200,-91.687,166.388,48.164,158.739
C03256=1023.411,-85.950,-91.697,166.391,48.161,158.738
C03257=1023.417,-85.701,-91.707,166.394,48.158,158.738
C03258=1023.424,-85.417,-91.718,166.397,48.154,158.738
C03259=1023.430,-85.134,-91.730,166.401,48.150,158.738
C03260=1023.437,-84.851,-91.741,166.404,48.146,158.738
C03261=1023.444,-84.568,-91.752,166.408,48.143,158.738
C03262=1023.449,-84.318,-91.762,166.411,48.139,158.737
C03263=1023.455,-84.068,-91.772,166.414,48.135,158.737
C03264=1023.461,-83.818,-91.783,166.417,48.132,158.737
C03265=1023.467,-83.568,-91.792,166.419,48.129,158.737
C03266=1023.472,-83.318,-91.803,166.423,48.125,158.737
C03267=1023.478,-83.069,-91.812,166.426,48.122,158.736
C03268=1023.484,-82.820,-91.823,166.429,48.118,158.736
C03269=1023.490,-82.570,-91.832,166.432,48.115,158.736
C03270=1023.495,-82.320,-91.842,166.435,48.111,158.736
C03271=1023.502,-82.071,-91.853,166.438,48.108,158.736
C03272=1023.507,-81.821,-91.863,166.441,48.104,158.735
C03273=1023.513,-81.571,-91.872,166.444,48.101,158.735
C03274=1023.519,-81.321,-91.883,166.447,48.098,158.735
C03275=1023.525,-81.071,-91.893,166.450,48.094,158.735
C03276=1023.531,-80.821,-91.903,166.453,48.091,158.735
C03277=1023.537,-80.572,-91.914,166.456,48.087,158.735
C03278=1023.543,-80.322,-91.923,166.459,48.084,158.734
C03279=1023.548,-80.072,-91.934,166.463,48.080,158.734
C03280=1023.555,-79.823,-91.944,166.465,48.077,158.734
C03281=1023.560,-79.573,-91.954,166.469,48.073,158.734
C03282=1023.566,-79.323,-91.965,166.472,48.070,158.734
C03283=1023.571,-79.073,-91.975,166.475,48.067,158.734
C03284=1023.577,-78.824,-91.986,166.477,48.064,158.733
C03285=1023.583,-78.574,-91.996,166.480,48.060,158.733
C03286=1023.589,-78.324,-92.006,166.483,48.057,158.733
C03287=1023.594,-78.074,-92.017,166.486,48.054,158.733
C03288=1023.600,-77.825,-92.027,166.490,48.051,158.733
C03289=1023.606,-77.575,-92.038,166.493,48.047,158.732
C03290=1023.612,-77.325,-92.048,166.496,48.044,158.732
C03291=1023.617,-77.075,-92.058,166.499,48.040,158.732
C03292=1023.623,-76.826,-92.069,166.502,48.037,158.732
C03293=1023.629,-76.576,-92.079,166.504,48.034,158.732
C03294=1023.634,-76.326,-92.090,166.507,48.030,158.732
C03295=1023.641,-76.077,-92.100,166.510,48.027,158.732
C03296=1023.646,-75.827,-92.110,166.514,48.024,158.731
C03297=1023.652,-75.577,-92.121,166.516,48.020,158.731
C03298=1023.657,-75.327,-92.131,166.520,48.017,158.731
C03299=1023.663,-75.078,-92.142,166.523,48.014,158.731
C03300=1023.670,-74.829,-92.153,166.526,48.011,158.731
C03301=1023.675,-74.579,-92.163,166.529,48.007,158.730
C03302=1023.681,-74.329,-92.174,166.532,48.004,158.730
C03303=1023.687,-74.080,-92.185,166.534,48.001,158.730
C03304=1023.692,-73.829,-92.195,166.537,47.997,158.730
C03305=1023.698,-73.580,-92.206,166.541,47.994,158.730
C03306=1023.703,-73.330,-92.216,166.544,47.991,158.730
C03307=1023.710,-73.080,-92.228,166.547,47.988,158.730
C03308=1023.715,-72.830,-92.238,166.549,47.985,158.729
C03309=1023.720,-72.580,-92.249,166.552,47.982,158.729
C03310=1023.726,-72.331,-92.260,166.556,47.979,158.729
C03311=1023.732,-72.081,-92.271,166.558,47.975,158.729
C03312=1023.737,-71.832,-92.282,166.562,47.972,158.729
C03313=1023.743,-71.582,-92.293,166.564,47.969,158.729
C03314=1023.749,-71.332,-92.303,166.567,47.965,158.728
C03315=1023.754,-71.083,-92.314,166.570,47.962,158.728
C03316=1023.760,-70.833,-92.325,166.573,47.959,158.728
C03317=1023.766,-70.583,-92.336,166.577,47.956,158.728
C03318=1023.772,-70.334,-92.347,166.580,47.953,158.728
C03319=1023.777,-70.084,-92.358,166.582,47.950,158.728
C03320=1023.783,-69.834,-92.369,166.585,47.947,158.728
C03321=1023.789,-69.585,-92.380,166.588,47.943,158.727
C03322=1023.796,-69.303,-92.392,166.591,47.940,158.727
C03323=1023.802,-69.022,-92.404,166.595,47.935,158.727
C03324=1023.808,-68.741,-92.417,166.598,47.932,158.727
C03325=1023.815,-68.460,-92.429,166.601,47.928,158.727
C03326=1023.820,-68.211,-92.440,166.604,47.925,158.726
C03327=1023.827,-67.960,-92.451,166.608,47.922,158.726
C03328=1023.832,-67.711,-92.462,166.611,47.919,158.726
C03329=1023.837,-67.461,-92.473,166.613,47.916,158.726
C03330=1023.843,-67.212,-92.484,166.616,47.913,158.726
C03331=1023.849,-66.962,-92.495,166.619,47.909,158.726
C03332=1023.855,-66.712,-92.506,166.622,47.906,158.725
C03333=1023.861,-66.462,-92.517,166.626,47.903,158.725
C03334=1023.867,-66.213,-92.528,166.629,47.899,158.725
C03335=1023.872,-65.963,-92.539,166.631,47.897,158.725
C03336=1023.879,-65.713,-92.550,166.634,47.893,158.725
C03337=1023.885,-65.464,-92.561,166.637,47.890,158.725
C03338=1023.890,-65.214,-92.572,166.640,47.886,158.724
C03339=1023.895,-64.964,-92.583,166.643,47.883,158.724
C03340=1023.902,-64.714,-92.595,166.647,47.880,158.724
C03341=1023.907,-64.465,-92.605,166.649,47.877,158.724
C03342=1023.913,-64.215,-92.616,166.652,47.874,158.724
C03343=1023.919,-63.966,-92.627,166.655,47.870,158.724
C03344=1023.925,-63.716,-92.638,166.658,47.867,158.723
C03345=1023.930,-63.466,-92.651,166.661,47.864,158.723
///RCONF 1,0,0,1,0,0,0,0,0,0,0,0,0,0,0,0,0,0,0,0,0,0,0,0
C03346=1023.936,-63.217,-92.662,166.663,47.861,158.723
C03347=1023.943,-62.967,-92.673,166.667,47.858,158.723
C03348=1023.948,-62.717,-92.684,166.670,47.854,158.723
C03349=1023.954,-62.468,-92.695,166.673,47.851,158.723
C03350=1023.960,-62.218,-92.706,166.676,47.847,158.722
C03351=1023.966,-61.968,-92.717,166.679,47.844,158.722
C03352=1023.971,-61.718,-92.728,166.681,47.841,158.722
C03353=1023.978,-61.469,-92.740,166.684,47.838,158.722
C03354=1023.983,-61.219,-92.751,166.687,47.834,158.722
C03355=1023.989,-60.970,-92.762,166.691,47.831,158.721
C03356=1023.996,-60.719,-92.773,166.694,47.828,158.721
C03357=1024.001,-60.470,-92.784,166.697,47.824,158.721
C03358=1024.007,-60.221,-92.796,166.699,47.821,158.721
C03359=1024.013,-59.971,-92.807,166.702,47.818,158.721
C03360=1024.019,-59.721,-92.818,166.705,47.815,158.721
C03361=1024.024,-59.472,-92.829,166.708,47.812,158.720
C03362=1024.031,-59.221,-92.840,166.711,47.808,158.720
C03363=1024.037,-58.973,-92.852,166.715,47.805,158.720
C03364=1024.043,-58.722,-92.863,166.717,47.802,158.720
C03365=1024.048,-58.473,-92.875,166.720,47.798,158.720
C03366=1024.054,-58.222,-92.886,166.723,47.795,158.719
C03367=1024.061,-57.974,-92.898,166.726,47.792,158.719
C03368=1024.066,-57.724,-92.908,166.729,47.789,158.719
C03369=1024.073,-57.474,-92.920,166.732,47.785,158.719
C03370=1024.079,-57.225,-92.931,166.735,47.782,158.719
C03371=1024.084,-56.974,-92.943,166.738,47.779,158.718
C03372=1024.090,-56.725,-92.954,166.741,47.776,158.718
C03373=1024.097,-56.475,-92.966,166.744,47.772,158.718
C03374=1024.102,-56.226,-92.977,166.747,47.768,158.718
C03375=1024.109,-55.976,-92.988,166.750,47.765,158.718
C03376=1024.114,-55.727,-93.000,166.753,47.761,158.717
C03377=1024.120,-55.477,-93.011,166.755,47.759,158.717
C03378=1024.126,-55.227,-93.022,166.758,47.755,158.717
C03379=1024.132,-54.978,-93.034,166.761,47.752,158.717
C03380=1024.139,-54.728,-93.045,166.764,47.748,158.717
C03381=1024.144,-54.478,-93.056,166.768,47.745,158.717
C03382=1024.150,-54.228,-93.069,166.771,47.742,158.716
C03383=1024.156,-53.979,-93.080,166.773,47.739,158.716
C03384=1024.163,-53.729,-93.091,166.776,47.735,158.716
C03385=1024.169,-53.479,-93.103,166.779,47.732,158.716
C03386=1024.176,-53.200,-93.116,166.782,47.728,158.715
C03387=1024.182,-52.919,-93.128,166.786,47.724,158.715
C03388=1024.189,-52.640,-93.141,166.789,47.720,158.715
C03389=1024.196,-52.360,-93.154,166.792,47.717,158.715
C03390=1024.201,-52.110,-93.166,166.795,47.713,158.715
C03391=1024.208,-51.860,-93.178,166.798,47.710,158.714
C03392=1024.214,-51.610,-93.189,166.801,47.707,158.714
C03393=1024.220,-51.361,-93.201,166.804,47.703,158.714
C03394=1024.227,-51.111,-93.212,166.807,47.700,158.714
C03395=1024.232,-50.862,-93.224,166.810,47.697,158.714
C03396=1024.238,-50.612,-93.235,166.812,47.693,158.713
C03397=1024.244,-50.362,-93.248,166.816,47.690,158.713
C03398=1024.250,-50.112,-93.259,166.819,47.687,158.713
C03399=1024.256,-49.863,-93.271,166.821,47.684,158.713
C03400=1024.261,-49.613,-93.284,166.824,47.681,158.713
C03401=1024.267,-49.363,-93.295,166.827,47.678,158.713
C03402=1024.273,-49.114,-93.307,166.831,47.675,158.712
C03403=1024.279,-48.864,-93.319,166.833,47.672,158.712
C03404=1024.285,-48.614,-93.331,166.836,47.669,158.712
C03405=1024.291,-48.365,-93.342,166.839,47.666,158.712
C03406=1024.297,-48.115,-93.355,166.841,47.662,158.712
C03407=1024.302,-47.866,-93.367,166.844,47.659,158.711
C03408=1024.309,-47.616,-93.378,166.848,47.656,158.711
C03409=1024.314,-47.366,-93.391,166.851,47.653,158.711
C03410=1024.321,-47.117,-93.402,166.853,47.650,158.711
C03411=1024.326,-46.867,-93.415,166.856,47.647,158.711
C03412=1024.331,-46.617,-93.427,166.859,47.643,158.711
C03413=1024.338,-46.368,-93.438,166.863,47.640,158.710
C03414=1024.344,-46.118,-93.451,166.864,47.637,158.710
C03415=1024.350,-45.869,-93.463,166.868,47.634,158.710
C03416=1024.356,-45.619,-93.475,166.871,47.630,158.710
C03417=1024.362,-45.369,-93.487,166.873,47.628,158.710
C03418=1024.368,-45.120,-93.499,166.876,47.624,158.709
C03419=1024.373,-44.870,-93.511,166.879,47.621,158.709
C03420=1024.380,-44.620,-93.523,166.883,47.618,158.709
C03421=1024.385,-44.371,-93.535,166.885,47.615,158.709
C03422=1024.391,-44.121,-93.548,166.888,47.611,158.709
C03423=1024.398,-43.871,-93.559,166.891,47.608,158.708
C03424=1024.403,-43.622,-93.571,166.894,47.605,158.708
C03425=1024.410,-43.372,-93.583,166.896,47.602,158.708
C03426=1024.416,-43.122,-93.596,166.900,47.599,158.708
C03427=1024.421,-42.873,-93.608,166.902,47.595,158.708
C03428=1024.427,-42.624,-93.620,166.906,47.592,158.708
C03429=1024.433,-42.374,-93.632,166.908,47.589,158.707
C03430=1024.440,-42.124,-93.644,166.911,47.586,158.707
C03431=1024.445,-41.875,-93.657,166.914,47.583,158.707
C03432=1024.451,-41.625,-93.669,166.916,47.579,158.707
C03433=1024.458,-41.375,-93.680,166.919,47.576,158.706
C03434=1024.464,-41.125,-93.693,166.923,47.573,158.706
C03435=1024.469,-40.876,-93.705,166.926,47.570,158.706
C03436=1024.475,-40.626,-93.717,166.928,47.567,158.706
C03437=1024.481,-40.376,-93.730,166.931,47.563,158.706
C03438=1024.488,-40.127,-93.742,166.934,47.560,158.706
C03439=1024.494,-39.877,-93.754,166.937,47.557,158.705
C03440=1024.499,-39.628,-93.766,166.939,47.554,158.705
C03441=1024.506,-39.378,-93.778,166.942,47.550,158.705
C03442=1024.512,-39.128,-93.791,166.946,47.547,158.705
C03443=1024.518,-38.878,-93.803,166.949,47.544,158.705
C03444=1024.524,-38.629,-93.816,166.951,47.541,158.704
C03445=1024.529,-38.379,-93.828,166.954,47.538,158.704
C03446=1024.535,-38.130,-93.841,166.956,47.535,158.704
C03447=1024.542,-37.881,-93.853,166.960,47.532,158.704
C03448=1024.548,-37.631,-93.866,166.963,47.529,158.704
C03449=1024.554,-37.381,-93.879,166.965,47.526,158.703
C03450=1024.560,-37.101,-93.893,166.969,47.522,158.703
C03451=1024.566,-36.821,-93.907,166.972,47.519,158.703
C03452=1024.573,-36.542,-93.920,166.975,47.515,158.703
C03453=1024.580,-36.263,-93.935,166.978,47.512,158.703
C03454=1024.586,-36.013,-93.947,166.981,47.509,158.703
C03455=1024.592,-35.763,-93.960,166.984,47.506,158.702
C03456=1024.598,-35.513,-93.973,166.987,47.503,158.702
C03457=1024.603,-35.265,-93.985,166.990,47.499,158.702
C03458=1024.609,-35.015,-93.998,166.992,47.496,158.702
C03459=1024.616,-34.765,-94.010,166.995,47.493,158.701
C03460=1024.622,-34.515,-94.023,166.997,47.490,158.701
C03461=1024.628,-34.266,-94.035,167.001,47.487,158.701
C03462=1024.634,-34.016,-94.048,167.004,47.484,158.701
C03463=1024.640,-33.766,-94.061,167.006,47.481,158.701
C03464=1024.646,-33.517,-94.073,167.009,47.478,158.701
C03465=1024.651,-33.268,-94.086,167.012,47.475,158.700
C03466=1024.657,-33.018,-94.099,167.014,47.471,158.700
C03467=1024.663,-32.768,-94.111,167.017,47.468,158.700
C03468=1024.669,-32.518,-94.124,167.021,47.465,158.700
C03469=1024.676,-32.269,-94.137,167.023,47.462,158.699
C03470=1024.682,-32.020,-94.149,167.026,47.459,158.699
C03471=1024.688,-31.770,-94.162,167.029,47.456,158.699
C03472=1024.694,-31.520,-94.175,167.031,47.452,158.699
C03473=1024.700,-31.270,-94.188,167.034,47.449,158.699
C03474=1024.706,-31.021,-94.200,167.038,47.446,158.699
C03475=1024.712,-30.771,-94.213,167.040,47.443,158.698
C03476=1024.718,-30.521,-94.226,167.043,47.440,158.698
C03477=1024.724,-30.272,-94.239,167.046,47.437,158.698
C03478=1024.730,-30.022,-94.252,167.048,47.433,158.698
C03479=1024.736,-29.772,-94.264,167.051,47.430,158.697
C03480=1024.742,-29.523,-94.278,167.055,47.427,158.697
C03481=1024.748,-29.273,-94.290,167.057,47.424,158.697
C03482=1024.754,-29.024,-94.302,167.060,47.421,158.697
C03483=1024.760,-28.775,-94.315,167.063,47.417,158.697
C03484=1024.766,-28.525,-94.328,167.065,47.415,158.696
C03485=1024.772,-28.276,-94.341,167.068,47.411,158.696
C03486=1024.778,-28.026,-94.353,167.071,47.408,158.696
C03487=1024.785,-27.776,-94.367,167.074,47.405,158.696
C03488=1024.791,-27.526,-94.380,167.077,47.402,158.696
C03489=1024.797,-27.277,-94.393,167.080,47.398,158.695
C03490=1024.803,-27.027,-94.405,167.082,47.396,158.695
C03491=1024.809,-26.778,-94.419,167.085,47.393,158.695
C03492=1024.815,-26.528,-94.432,167.088,47.389,158.695
C03493=1024.821,-26.278,-94.445,167.091,47.387,158.695
C03494=1024.827,-26.029,-94.458,167.094,47.383,158.694
C03495=1024.833,-25.779,-94.471,167.096,47.381,158.694
C03496=1024.839,-25.530,-94.484,167.099,47.377,158.694
C03497=1024.844,-25.280,-94.497,167.102,47.374,158.694
C03498=1024.850,-25.031,-94.511,167.105,47.371,158.694
C03499=1024.856,-24.781,-94.523,167.108,47.368,158.694
C03500=1024.863,-24.531,-94.536,167.110,47.366,158.693
C03501=1024.869,-24.282,-94.550,167.113,47.362,158.693
C03502=1024.874,-24.032,-94.563,167.115,47.359,158.693
C03503=1024.880,-23.783,-94.576,167.118,47.356,158.693
C03504=1024.886,-23.533,-94.589,167.122,47.353,158.692
C03505=1024.892,-23.284,-94.602,167.124,47.350,158.692
C03506=1024.899,-23.034,-94.615,167.127,47.347,158.692
C03507=1024.904,-22.785,-94.629,167.129,47.344,158.692
C03508=1024.910,-22.535,-94.642,167.132,47.341,158.692
C03509=1024.916,-22.286,-94.655,167.136,47.338,158.692
C03510=1024.923,-22.036,-94.669,167.138,47.335,158.691
C03511=1024.928,-21.786,-94.682,167.141,47.332,158.691
C03512=1024.934,-21.536,-94.695,167.143,47.328,158.691
C03513=1024.941,-21.287,-94.708,167.146,47.325,158.691
C03514=1024.948,-21.007,-94.723,167.149,47.322,158.690
C03515=1024.954,-20.726,-94.738,167.152,47.318,158.690
C03516=1024.961,-20.446,-94.752,167.155,47.315,158.690
C03517=1024.968,-20.165,-94.768,167.158,47.311,158.690
C03518=1024.976,-19.809,-94.787,167.162,47.307,158.689
C03519=1024.985,-19.453,-94.806,167.166,47.302,158.689
C03520=1024.991,-19.203,-94.819,167.169,47.299,158.689
C03521=1024.997,-18.953,-94.832,167.172,47.296,158.689
C03522=1025.004,-18.704,-94.846,167.175,47.293,158.688
C03523=1025.010,-18.454,-94.859,167.178,47.290,158.688
C03524=1025.016,-18.205,-94.873,167.180,47.287,158.688
C03525=1025.021,-17.955,-94.886,167.183,47.284,158.688
C03526=1025.027,-17.706,-94.899,167.186,47.280,158.688
C03527=1025.034,-17.456,-94.912,167.188,47.278,158.687
C03528=1025.040,-17.206,-94.926,167.192,47.275,158.687
C03529=1025.046,-16.957,-94.940,167.194,47.271,158.687
C03530=1025.052,-16.707,-94.953,167.197,47.268,158.687
C03531=1025.058,-16.458,-94.966,167.200,47.265,158.687
C03532=1025.065,-16.208,-94.980,167.202,47.262,158.686
C03533=1025.070,-15.958,-94.993,167.205,47.259,158.686
C03534=1025.077,-15.709,-95.006,167.207,47.255,158.686
C03535=1025.083,-15.460,-95.020,167.210,47.252,158.686
C03536=1025.088,-15.210,-95.034,167.213,47.249,158.685
C03537=1025.095,-14.960,-95.047,167.216,47.246,158.685
C03538=1025.101,-14.710,-95.061,167.219,47.243,158.685
C03539=1025.107,-14.461,-95.074,167.221,47.240,158.685
C03540=1025.112,-14.212,-95.088,167.225,47.237,158.685
C03541=1025.119,-13.962,-95.102,167.227,47.234,158.684
C03542=1025.125,-13.712,-95.116,167.230,47.231,158.684
C03543=1025.131,-13.463,-95.130,167.232,47.228,158.684
C03544=1025.137,-13.214,-95.143,167.235,47.225,158.684
C03545=1025.143,-12.964,-95.157,167.238,47.223,158.684
C03546=1025.149,-12.714,-95.171,167.241,47.219,158.683
C03547=1025.155,-12.465,-95.184,167.243,47.217,158.683
C03548=1025.161,-12.215,-95.198,167.246,47.213,158.683
C03549=1025.167,-11.965,-95.212,167.248,47.211,158.683
C03550=1025.173,-11.716,-95.226,167.251,47.207,158.682
C03551=1025.179,-11.467,-95.239,167.254,47.204,158.682
C03552=1025.185,-11.217,-95.253,167.257,47.201,158.682
C03553=1025.192,-10.968,-95.267,167.259,47.198,158.682
C03554=1025.197,-10.718,-95.281,167.262,47.195,158.682
C03555=1025.203,-10.469,-95.294,167.264,47.192,158.681
C03556=1025.209,-10.219,-95.308,167.268,47.189,158.681
C03557=1025.216,-9.969,-95.322,167.271,47.186,158.681
C03558=1025.221,-9.720,-95.336,167.273,47.183,158.681
C03559=1025.228,-9.470,-95.349,167.276,47.180,158.681
C03560=1025.234,-9.221,-95.364,167.278,47.177,158.680
C03561=1025.240,-8.972,-95.377,167.281,47.173,158.680
C03562=1025.246,-8.721,-95.391,167.284,47.171,158.680
C03563=1025.251,-8.472,-95.405,167.287,47.167,158.680
C03564=1025.258,-8.222,-95.418,167.289,47.165,158.680
C03565=1025.264,-7.973,-95.433,167.292,47.162,158.679
C03566=1025.270,-7.724,-95.447,167.294,47.159,158.679
C03567=1025.276,-7.474,-95.461,167.297,47.155,158.679
C03568=1025.283,-7.224,-95.474,167.299,47.152,158.679
C03569=1025.288,-6.975,-95.489,167.303,47.149,158.678
C03570=1025.295,-6.725,-95.502,167.305,47.146,158.678
C03571=1025.301,-6.475,-95.516,167.308,47.143,158.678
C03572=1025.307,-6.226,-95.530,167.311,47.140,158.678
C03573=1025.313,-5.977,-95.544,167.313,47.137,158.677
C03574=1025.319,-5.727,-95.558,167.316,47.133,158.677
C03575=1025.326,-5.477,-95.572,167.319,47.131,158.677
C03576=1025.334,-5.124,-95.592,167.322,47.126,158.677
C03577=1025.343,-4.770,-95.612,167.326,47.122,158.676
C03578=1025.351,-4.417,-95.631,167.330,47.117,158.676
C03579=1025.360,-4.063,-95.651,167.334,47.113,158.676
C03580=1025.366,-3.813,-95.666,167.337,47.110,158.676
///RCONF 1,0,0,0,0,0,0,0,0,0,0,0,0,0,0,0,0,0,0,0,0,0,0,0
C03581=1025.373,-3.564,-95.679,167.339,47.107,158.675
C03582=1025.378,-3.315,-95.693,167.342,47.104,158.675
C03583=1025.384,-3.065,-95.708,167.345,47.101,158.675
C03584=1025.390,-2.815,-95.722,167.347,47.098,158.675
C03585=1025.396,-2.566,-95.737,167.350,47.095,158.675
C03586=1025.402,-2.316,-95.751,167.352,47.093,158.674
